930: // Query Input Value Occupancy
	IF (_bEnablePushButton) THEN
		fb301PushButton(	bInitialize := FALSE,
								bQueryInputValue := TRUE,
								bGetInputNotifications := FALSE,
								nShortAddress := nShortAddress,
								nInstanceNumber := 0);
		IF (NOT fb301PushButton.bReadingInputValue) THEN
			nPushBotton := fb301PushButton.nPushButtonEvent;
			nStep := 940;
			fb301PushButton(bInitialize := FALSE, bQueryInputValue := FALSE);
		END_IF
	ELSE
		nPushBotton := 1;
		nStep := 940;
	END_IF

940: // Query Input Value rotation direction
	IF (_bEnableRotation) THEN
		fb301Rotation(
			bInitialize:= FALSE, 
			nShortAddress:= nShortAddress, 
			nInstanceNumber:= 1, 
			bQueryInputValue:= TRUE, 
			bGetInputNotifications:= FALSE);	 
	
		IF (NOT fb301Rotation.bReadingInputValue) THEN
			nRotation := 4 ;//fb301Rotation.nPushButtonEvent; This are disabled, due to no data to query, before the device has being rotated
			nStep := 950;
			fb301Rotation(bQueryInputValue := FALSE);
		END_IF
	ELSE
		nRotation := 4;
		nStep := 950;
	END_IF

950: // Query Input actual position
	IF (_bEnablePosition) THEN
		fb302AbsoluteInputDevice(	bInitialize := FALSE,
							bQueryInputValue := TRUE,
							nShortAddress := nShortAddress,
							nInstanceNumber := 2,
							nResolution := 8);
		IF (NOT fb302AbsoluteInputDevice.bReadingInputValue) THEN
			nPosition := fb302AbsoluteInputDevice.nInputLevel;
			nStep := 0;
			fb302AbsoluteInputDevice(bInitialize := FALSE, bQueryInputValue := FALSE);
		END_IF
	ELSE
		nPosition := 0;
		nStep := 0;
	END_IF
{endregion}

ELSE
	nStep := 0;
END_CASE

THIS^.SetCommunication();
IF (THIS^.ParameterChanged()) THEN
	nErrorId := THIS^.CheckParameters();
	bError := (nErrorId > 0);
	IF (bError) THEN
		bParameterInvalid := TRUE;
		RETURN;
	ELSE
		bParameterInvalid := FALSE;
	END_IF
END_IF
IF (bParameterInvalid) THEN
	RETURN;
END_IF

{region 'Notifications'}
IF (NOT bInitializing) THEN
	rtrigReadingPushBotton(CLK := bQueryPushBotton);
	IF (rtrigReadingPushBotton.Q) THEN
		bReadingPushbotton:= TRUE;
	END_IF
	rtrigReadingRotation(CLK := bQueryRotation);
	IF (rtrigReadingRotation.Q) THEN
		bReadingRotation := TRUE;
	END_IF
	rtrigReadingPosition(CLK := bQueryPosition);
	IF (rtrigReadingPosition.Q) THEN
		bReadingPosition := TRUE;
	END_IF

	THIS^.SetCommunication();

	fb103ControlDevice(	bInitialize := FALSE,
						bGetPowerCycleNotifications := FALSE,
						nShortAddress := nShortAddress);
	rtrigError103Generic(CLK := fb103ControlDevice.bError);
	ftrigError103Generic(CLK := fb103ControlDevice.bError);
	IF (rtrigError103Generic.Q OR ftrigError103Generic.Q) THEN
		nErrorId := fb103ControlDevice.ipResultMessage.nEventId;
		bError := fb103ControlDevice.bError;
	END_IF

{region 'Pushbotton'}
	fb301PushButton(
		bInitialize:= FALSE, 
		nShortAddress:= nShortAddress, 
		nInstanceNumber:= 0, 
		bQueryInputValue:= bQueryPushBotton, 
		bGetInputNotifications:= TRUE);

	IF (bReadingPushbotton) THEN
		IF (NOT fb301PushButton.bReadingInputValue) THEN
			bReadingPushbotton := FALSE;
			IF (NOT fb301PushButton.bError) THEN
				nPushBotton := fb301PushButton.nPushButtonEvent;
			END_IF
		END_IF
	END_IF
	IF (NOT fb301PushButton.bError) THEN
		nPushBotton := fb301PushButton.nPushButtonEvent;
	END_IF
	rtrigError301PushButton(CLK := fb301PushButton.bError);
	ftrigError301PushButton(CLK := fb301PushButton.bError);
	IF (rtrigError301PushButton.Q OR ftrigError301PushButton.Q) THEN
		nErrorId := fb301PushButton.ipResultMessage.nEventId;
		bError := fb301PushButton.bError;
	END_IF
{endregion}

{region 'Rotation'}
	 
	fb301Rotation(
		bInitialize:= FALSE, 
		nShortAddress:= nShortAddress, 
		nInstanceNumber:= 1, 
		bQueryInputValue:= bQueryRotation, 
		bGetInputNotifications:= TRUE);	 		   
						 
	IF (bReadingRotation) THEN
		IF (NOT fb301Rotation.bReadingInputValue) THEN
			bReadingRotation := FALSE;
			IF (NOT fb301Rotation.bError) THEN
				nRotation := fb301Rotation.nPushButtonEvent;
			END_IF
		END_IF
	END_IF
	IF (NOT fb301Rotation.bError) THEN
		nRotation := fb301Rotation.nPushButtonEvent;
	END_IF
	rtrigError301Rotation(CLK := fb301Rotation.bError);
	ftrigError301Rotation(CLK := fb301Rotation.bError);
	IF (rtrigError301Rotation.Q OR ftrigError301Rotation.Q) THEN
		nErrorId := fb301Rotation.ipResultMessage.nEventId;
		bError := fb301Rotation.bError;
	END_IF
{endregion}

{region 'Position'}
	fb302AbsoluteInputDevice( bInitialize:= FALSE, 
						nShortAddress:= , 
						nInstanceNumber:= 2, 
						nResolution:= 8, 
						bQueryInputValue:= bQueryPosition, 
						bGetInputNotifications:= TRUE);

	IF (bReadingPosition) THEN
		IF (NOT fb302AbsoluteInputDevice.bReadingInputValue) THEN
			bReadingPosition := FALSE;
			IF (NOT fb302AbsoluteInputDevice.bError) THEN
				nPosition := fb302AbsoluteInputDevice.nInputLevel;
			END_IF
		END_IF
	END_IF
	IF (NOT fb302AbsoluteInputDevice.bError) THEN
		nPosition := fb302AbsoluteInputDevice.nInputLevel;
	END_IF
	rtrigError302AbsoluteInputDevice(CLK := fb302AbsoluteInputDevice.bError);
	ftrigError302AbsoluteInputDevice(CLK := fb302AbsoluteInputDevice.bError);
	IF (rtrigError302AbsoluteInputDevice.Q OR ftrigError302AbsoluteInputDevice.Q) THEN
		nErrorId := fb302AbsoluteInputDevice.ipResultMessage.nEventId;
		bError := fb302AbsoluteInputDevice.bError;
	END_IF
{endregion}
		  
END_IF
{endregion}

IF (bError) THEN
	nPushBotton := 1;
	nRotation := 4;
	nPosition := 0;
END_IF

IF nPushBotton.0 THEN
	bPressed := FALSE;
	bReleased:= TRUE;
END_IF
IF nPushBotton.1 THEN
	bPressed := TRUE;
	bReleased:= FALSE;
END_IF

IF nRotation.2 THEN
	bNeutral:= TRUE;
	bCCW := FALSE;
	bCW := FALSE;
ELSIF nRotation.0 THEN
	bNeutral:= FALSE;
	bCCW := FALSE;
	bCW := TRUE;
ELSIF nRotation.1 THEN
	bNeutral:= FALSE;
	bCCW := TRUE;
	bCW := FALSE;	
END_IF

stROTdata.bStopped:= bNeutral ;
stROTdata.bCW:= bCW ;
stROTdata.bCCW:= bCCW ;
stROTdata.bPressed:= bPressed ;
stROTdata.bReleased:= bReleased ;
stROTdata.nPos:= LWORD_TO_BYTE(nPosition) ;

// A TRUE at this input enables the instance for detecting movement. A FALSE at this input causes the sending of events from this instance to be disabled.
{attribute 'monitoring' := 'call'}
PROPERTY PUBLIC bEnablePosition : BOOL
GET
bEnablePosition := _bEnablePosition;
END_GET
SET
_bEnablePosition := bEnablePosition;
END_SET
END_PROPERTY

// Setting of the event priority (Low, MiddleLow, Middle, MiddleHigh).
{attribute 'monitoring' := 'call'}
PROPERTY PUBLIC eEventPriorityPosition : E_DALIEventPriority
GET
eEventPriorityPosition := _eEventPriorityPosition;
END_GET
SET
_eEventPriorityPosition := eEventPriorityPosition;
END_SET
END_PROPERTY

// Dead time (0...12750 ms) to ensure that not too many events are sent in succession. An event is only sent after expiry of the dead time timer. The dead time timer is restarted each time an event is sent.
{attribute 'monitoring' := 'call'}
PROPERTY PUBLIC nDeadtimerPosition : UINT
GET
nDeadtimerPosition := _nDeadtimeTimerPosition;
END_GET
SET
_nDeadtimeTimerPosition := nDeadtimerPosition;
END_SET
END_PROPERTY

// Time (0…255 s) after which the pending event of the measurement is repeated if no other event has occurred in the meantime.
{attribute 'monitoring' := 'call'}
PROPERTY PUBLIC nReportTimePosition : BYTE
GET
nReportTimePosition := _nReportTimerPosition;
END_GET
SET
_nReportTimerPosition := nReportTimePosition;
END_SET
END_PROPERTY

// A TRUE at this input enables the instance for measuring the brightness. A FALSE at this input causes the sending of events from this instance to be disabled.
{attribute 'monitoring' := 'call'}
PROPERTY PUBLIC bEnablePushButton : BOOL
GET
bEnablePushButton := _bEnablePushButton;
END_GET
SET
_bEnablePushButton := bEnablePushButton;
END_SET
END_PROPERTY

// Setting of the event priority (Low, MiddleLow, Middle, MiddleHigh).
{attribute 'monitoring' := 'call'}
PROPERTY PUBLIC eEventPriorityButton : E_DALIEventPriority
GET
eEventPriorityButton := _eEventPriorityPushButton;
END_GET
SET
_eEventPriorityPushButton := eEventPriorityButton;
END_SET
END_PROPERTY

// Deadtime (0...12750 ms), to ensure to send out an event until the deadtime timer has expired. The deadtime timer will be restarted every time an event is sent.
{attribute 'monitoring' := 'call'}
PROPERTY PUBLIC nDoubleTimerPushButton : UINT
GET
nDoubleTimerPushButton := _nDoubleTimerPushButton;
END_GET
SET
_nDoubleTimerPushButton := nDoubleTimerPushButton;
END_SET
END_PROPERTY

// Time (0...255 s) after which the pending event of the brightness sensor is repeated if no other event has occurred in the meantime.
{attribute 'monitoring' := 'call'}
PROPERTY PUBLIC nEventFilterPushButton : BYTE
GET
nEventFilterPushButton := _nEventFilterPushButton;
END_GET
SET
_nEventFilterPushButton := nEventFilterPushButton;
END_SET
END_PROPERTY

// Value (0...25 %) for calculating a hysteresis value in order to prevent frequent and disturbing changes when measuring the brightness.
{attribute 'monitoring' := 'call'}
PROPERTY PUBLIC nRepeatTimerPushButton : uint
GET
nRepeatTimerPushButton := _nRepeatTimerPushButton;
END_GET
SET
_nRepeatTimerPushButton := nRepeatTimerPushButton;
END_SET
END_PROPERTY

// As the percentage hysteresis can also lead to large fluctuations at low brightness, a minimum hysteresis (0...255) can be specified with this variable.
{attribute 'monitoring' := 'call'}
PROPERTY PUBLIC nShortTimerPushButton : UINT
GET
nShortTimerPushButton := _nShortTimerPushButton;
END_GET
SET
_nShortTimerPushButton := nShortTimerPushButton;
END_SET
END_PROPERTY

// Time (0...255 s) after which the pending event of the brightness sensor is repeated if no other event has occurred in the meantime.
{attribute 'monitoring' := 'call'}
PROPERTY PUBLIC nStuckTimerPushButton : BYTE
GET
nStuckTimerPushButton := _nStuckTimerPushButton;
END_GET
SET
_nStuckTimerPushButton := nStuckTimerPushButton;
END_SET
END_PROPERTY

// A TRUE at this input enables the instance for detecting movement. A FALSE at this input causes the sending of events from this instance to be disabled.
{attribute 'monitoring' := 'call'}
PROPERTY PUBLIC bEnableRotation : BOOL
GET
bEnableRotation := _bEnableRotation;
END_GET
SET
_bEnableRotation := bEnableRotation;
END_SET
END_PROPERTY

// Setting of the event priority (Low, MiddleLow, Middle, MiddleHigh).
{attribute 'monitoring' := 'call'}
PROPERTY PUBLIC eEventPriorityRotation : E_DALIEventPriority
GET
eEventPriorityRotation := _eEventPriorityRotation;
END_GET
SET
_eEventPriorityRotation := eEventPriorityRotation;
END_SET
END_PROPERTY

// Setting of the event filter.
{attribute 'monitoring' := 'call'}
PROPERTY PUBLIC nEventFilterRotation : byte
GET
nEventFilterRotation := _nEventFilterRotation;
END_GET
SET
_nEventFilterRotation:= nEventFilterRotation;
END_SET
END_PROPERTY

// Checks whether all parameters are valid.
// Return codes:
//   0: no error.
//	 1..999: error codes of the library
//   1000... : custom error codes
METHOD PRIVATE CheckParameters : UDINT
CheckParameters := 0;
IF (_ipDALICommunication = 0) THEN
	CheckParameters := TC_EVENTS.TcDALIEventClass.TheInterfaceToTheCommunicationBufferIsNotInitialized.nEventId;
ELSIF (nShortAddress > 63) THEN
	CheckParameters := TC_EVENTS.TcDALIEventClass.ParameterShortAddressLiesOutsideOfTheValidRange2.nEventId;
{region 'Botton'}
ELSIF (_nDoubleTimerPushButton > 2000) THEN
	CheckParameters := TC_EVENTS.TcDALIEventClass.ParameterDoubleTimerPart301LiesOutsideOfTheValidRange.nEventId;
ELSIF ((_nRepeatTimerPushButton < 100) OR (_nRepeatTimerPushButton > 2000)) THEN
	CheckParameters := TC_EVENTS.TcDALIEventClass.ParameterRepeatTimerLiesOutsideOfTheValidRange.nEventId;
ELSIF (nShortTimerPushButton > 5100) THEN
	CheckParameters := TC_EVENTS.TcDALIEventClass.ParameterShortTimerPart301LiesOutsideOfTheValidRange.nEventId;
ELSIF ((_nStuckTimerPushButton < 5) OR (_nStuckTimerPushButton > 255)) THEN
	CheckParameters := TC_EVENTS.TcDALIEventClass.ParameterStuckTimerPart301LiesOutsideOfTheValidRange.nEventId;
ELSIF ((_eEventPriorityPushButton <> E_DALIEventPriority.Low) AND (_eEventPriorityPushButton <> E_DALIEventPriority.MiddleLow) AND
       (_eEventPriorityPushButton <> E_DALIEventPriority.Middle) AND (_eEventPriorityPushButton <> E_DALIEventPriority.MiddleHigh)) THEN
	CheckParameters := TC_EVENTS.TcDALIEventClass.ParameterEventPriorityDeviceLiesOutsideOfTheValidRange.nEventId;
{endregion}
{region 'Rotation'}
ELSIF ((_eEventPriorityRotation <> E_DALIEventPriority.Low) AND (_eEventPriorityRotation <> E_DALIEventPriority.MiddleLow) AND
       (_eEventPriorityRotation <> E_DALIEventPriority.Middle) AND (_eEventPriorityRotation <> E_DALIEventPriority.MiddleHigh)) THEN
	CheckParameters := TC_EVENTS.TcDALIEventClass.ParameterEventPriorityDeviceLiesOutsideOfTheValidRange.nEventId;
{endregion}
{region 'Position'}
ELSIF (_nDeadtimeTimerPosition > 12750) THEN
	CheckParameters := TC_EVENTS.TcDALIEventClass.ParameterDeadtimeTimerPart302LiesOutsideOfTheValidRange.nEventId;
ELSIF ((_eEventPriorityPosition <> E_DALIEventPriority.Low) AND (_eEventPriorityPosition <> E_DALIEventPriority.MiddleLow) AND
       (_eEventPriorityPosition <> E_DALIEventPriority.Middle) AND (_eEventPriorityPosition <> E_DALIEventPriority.MiddleHigh)) THEN
	CheckParameters := TC_EVENTS.TcDALIEventClass.ParameterEventPriorityDeviceLiesOutsideOfTheValidRange.nEventId;
{endregion}
//ELSIF (check your parameter) THEN
//	CheckParameters := 1000;
//ELSIF (check another parameter) THEN
//	CheckParameters := 1001;
END_IF
END_METHOD

METHOD FB_init : BOOL
VAR_INPUT
	bInitRetains			:	BOOL; // if TRUE, the retain variables are initialized (warm start / cold start)
	bInCopyCode				:	BOOL;  // if TRUE, the instance afterwards gets moved into the copy code (online change)
	ipDALICommunication 	:	I_DALICommunication;
END_VAR
_ipDALICommunication := ipDALICommunication;
END_METHOD

// Property to set the referenz to the communication function block.
{attribute 'monitoring' := 'call'}
PROPERTY PUBLIC ipDALICommunication : I_DALICommunication
GET
ipDALICommunication := _ipDALICommunication;
END_GET
SET
_ipDALICommunication := ipDALICommunication;
END_SET
END_PROPERTY

// Return codes:
//   FALSE: no change
//   TRUE: parameter are changed
{attribute 'hide'}
METHOD PRIVATE ParameterChanged : BOOL
VAR_INPUT
END_VAR
IF (nShortAddress <> nShortAddressCheck) THEN
	ParameterChanged := TRUE;
	nShortAddressCheck := nShortAddress;
ELSE
	ParameterChanged := FALSE;
END_IF
END_METHOD

// Apply the preset value of IpDALICommunication if available.
METHOD PRIVATE SetCommunication : BOOL
VAR_INPUT
END_VAR
fb103ControlDevice.ipDALICommunication := THIS^.ipDALICommunication;
fb301PushButton.ipDALICommunication := THIS^.ipDALICommunication;
fb301Rotation.ipDALICommunication := THIS^.ipDALICommunication;
fb302AbsoluteInputDevice.ipDALICommunication := THIS^.ipDALICommunication;
fbSavePersistentVariables.ipDALICommunication := THIS^.ipDALICommunication;
fbStartQuiescentMode.ipDALICommunication := THIS^.ipDALICommunication;
fbStopQuiescentMode.ipDALICommunication := THIS^.ipDALICommunication;
END_METHOD

END_FUNCTION_BLOCK

// POUs/DALI/DALI_Devices/Lunatone/FB_DALI_LunatoneMC
FUNCTION_BLOCK FB_DALI_LunatoneMC
VAR_INPUT
	byShrtAdr				: BYTE;
	bInitialize				: BOOL := TRUE;
	ipCommunication			: I_DALICommunication;
	DALI_LINE_NUM			: INT := 1;	
	stLunatoneMCSetup		: ST_LunatoneMCSetup;		
END_VAR
VAR_OUTPUT
	arrButtons				: ARRAY [1..4] OF ST_DALIButton;
END_VAR
		
VAR
	fbButtons 				: FB_DALI_Lunatone_MC(0) ;

	arrQueryInput 			: ARRAY [1..4] OF BOOL;
	arrReadingInput 		: ARRAY [1..4] OF BOOL;
	arrPushButtonEvent 		: ARRAY [1..4] OF WORD; (* Bit 0 - Push button released.
									 Bit 1 - Push button pressed..
									 Bit 2 - Short keystroke.
									 Bit 3 - Double keystroke.
									 Bit 4 - Start long keystroke.
									 Bit 5 - Repeat long keystroke.
									 Bit 6 - Stop long keystroke.
									 Bit 7 - Push button free again; was previously blocked.
									 Bit 8 - Push button blocked. *)

	fbDelaySetupDALIDevice	: TON;
	tDelayTime				: TIME;
	bInitSensor				: BOOL;
	fbInitDone				: F_TRIG;
	bInitDone				: BOOL;
	bInitErr				: BOOL;
	bInitializing			: BOOL;
	bInitTimeOut			: BOOL;
	fbInitTimeOut			: TON;
END_VAR

fbButtons.ipDALICommunication:= ipCommunication ;

	fbButtons.bEnablePushButton1:= stLunatoneMCSetup.arrEnablePushButton[1];
	fbButtons.bEnablePushButton2:= stLunatoneMCSetup.arrEnablePushButton[2];
	fbButtons.bEnablePushButton3:= stLunatoneMCSetup.arrEnablePushButton[3];
	fbButtons.bEnablePushButton4:= stLunatoneMCSetup.arrEnablePushButton[4];
	
	fbButtons.eEventPriorityPushButton1:= stLunatoneMCSetup.arrEventPriorityPushButton[1];
	fbButtons.eEventPriorityPushButton2:= stLunatoneMCSetup.arrEventPriorityPushButton[2];
	fbButtons.eEventPriorityPushButton3:= stLunatoneMCSetup.arrEventPriorityPushButton[3];
	fbButtons.eEventPriorityPushButton4:= stLunatoneMCSetup.arrEventPriorityPushButton[4];

	fbButtons.nDoubleTimerPushButton1 := stLunatoneMCSetup.nDoubleTimerPushButton;
	fbButtons.nDoubleTimerPushButton2:= stLunatoneMCSetup.nDoubleTimerPushButton;
	fbButtons.nDoubleTimerPushButton3:= stLunatoneMCSetup.nDoubleTimerPushButton;
	fbButtons.nDoubleTimerPushButton4:= stLunatoneMCSetup.nDoubleTimerPushButton;
	
	fbButtons.nEventFilterPushButton1 :=stLunatoneMCSetup.nEventFilterPushButton[1] ;
	fbButtons.nEventFilterPushButton2 :=stLunatoneMCSetup.nEventFilterPushButton[2] ;
	fbButtons.nEventFilterPushButton3 :=stLunatoneMCSetup.nEventFilterPushButton[3] ;
	fbButtons.nEventFilterPushButton4 :=stLunatoneMCSetup.nEventFilterPushButton[4] ;
	
	fbButtons.nRepeatTimerPushButton1 := stLunatoneMCSetup.nRepeatTimerPushButton;
	fbButtons.nRepeatTimerPushButton2 := stLunatoneMCSetup.nRepeatTimerPushButton;
	fbButtons.nRepeatTimerPushButton3 := stLunatoneMCSetup.nRepeatTimerPushButton;
	fbButtons.nRepeatTimerPushButton4 := stLunatoneMCSetup.nRepeatTimerPushButton;
	
	fbButtons.nShortTimerPushButton1 := stLunatoneMCSetup.nShortTimerPushButton ;
	fbButtons.nShortTimerPushButton2 := stLunatoneMCSetup.nShortTimerPushButton ;
	fbButtons.nShortTimerPushButton3 := stLunatoneMCSetup.nShortTimerPushButton ;
	fbButtons.nShortTimerPushButton4 := stLunatoneMCSetup.nShortTimerPushButton ;
	
	fbButtons.nStuckTimerPushButton1 := stLunatoneMCSetup.nStuckTimerPushButton ;
	fbButtons.nStuckTimerPushButton2 := stLunatoneMCSetup.nStuckTimerPushButton ;
	fbButtons.nStuckTimerPushButton3 := stLunatoneMCSetup.nStuckTimerPushButton ;
	fbButtons.nStuckTimerPushButton4 := stLunatoneMCSetup.nStuckTimerPushButton ;

//Calculate delay time for init sensor
tDelayTime := INT_TO_TIME((BYTE_TO_INT(byShrtAdr) * 400));	
fbDelaySetupDALIDevice(IN:= bInitialize , PT:=tDelayTime , Q=> , ET=> );	
	
IF fbDelaySetupDALIDevice.q AND NOT GVL_DALI.arrbBlockDTR[DALI_LINE_NUM] AND NOT (bInitDone OR bInitErr) THEN
	bInitDone := FALSE;
	bInitErr := FALSE;
	bInitSensor:= TRUE;
	GVL_DALI.arrbBlockDTR[DALI_LINE_NUM]:= TRUE;
END_IF

fbButtons(
	bError=> , 
	ipResultMessage=> , 
	bInitialize:= bInitSensor , 
	nShortAddress:= byShrtAdr, 
	nOptions:= , 
	bQueryInputValue1:= arrQueryInput[1], 
	bQueryInputValue2:= arrQueryInput[2], 
	bQueryInputValue3:= arrQueryInput[3], 
	bQueryInputValue4:= arrQueryInput[4], 
	bInitializing=> bInitializing, 
	bReadingInputValue1=> arrReadingInput[1] , 
	bReadingInputValue2=> arrReadingInput[2] , 
	bReadingInputValue3=> arrReadingInput[3] , 
	bReadingInputValue4=> arrReadingInput[4] , 
	nPushButton1Event=> arrPushButtonEvent[1], 
	nPushButton2Event=> arrPushButtonEvent[2], 
	nPushButton3Event=> arrPushButtonEvent[3], 
	nPushButton4Event=> arrPushButtonEvent[4]
);	
fbInitDone(CLK:=bInitSensor AND bInitializing );	
	IF fbInitDone.Q THEN
		IF NOT bInitTimeOut THEN
			bInitDone := TRUE;
			bInitErr := FALSE;
			GVL_DALI.arrbBlockDTR[DALI_LINE_NUM]:= FALSE;
		ELSE
			bInitErr := TRUE;
			GVL_DALI.arrbBlockDTR[DALI_LINE_NUM]:= FALSE;
		END_IF
	END_IF

fbInitTimeOut(IN:=bInitializing, PT:= T#15S); 

IF fbInitTimeOut.Q THEN
	bInitErr := TRUE;
	GVL_DALI.arrbBlockDTR[DALI_LINE_NUM]:= FALSE;
END_IF


IF NOT bInitialize THEN
		fbInitTimeOut(IN:= FALSE);
		bInitSensor:= FALSE;
		bInitDone := FALSE;
		bInitErr := FALSE;
END_IF	
	A_Sort_Event_Button1();
	A_Sort_Event_Button2();
	A_Sort_Event_Button3();
	A_Sort_Event_Button4();

ACTION A_Sort_Event_Button1:
IF arrPushButtonEvent[1].1 THEN
	arrButtons[1].bPressed:= TRUE;
	arrButtons[1].bReleased:= FALSE;
END_IF

IF arrPushButtonEvent[1].0 THEN
	arrButtons[1].bPressed:= FALSE;
	arrButtons[1].bReleased:= TRUE;
END_IF

IF arrPushButtonEvent[1].2 THEN
	arrButtons[1].bShortPress:= TRUE;
END_IF

IF arrPushButtonEvent[1].3 THEN
	arrButtons[1].bDoublePress:= TRUE;
END_IF

IF arrPushButtonEvent[1].4 THEN
	arrButtons[1].bLongPressStop:= FALSE;
	arrButtons[1].bLongPressStart:= TRUE;
	arrButtons[1].bLongPressRepeat:= FALSE;	
END_IF

arrButtons[1].bLongPressRepeat:= arrPushButtonEvent[1].5 ;

IF arrPushButtonEvent[1].6 THEN
	arrButtons[1].bLongPressStop:= TRUE;
	arrButtons[1].bLongPressStart:= FALSE;
	arrButtons[1].bLongPressRepeat:= FALSE;	
END_IF

IF arrPushButtonEvent[1].7 THEN
	arrButtons[1].bPressed:= FALSE;
	arrButtons[1].bReleased:= FALSE;
	arrButtons[1].bShortPress:= FALSE;
	arrButtons[1].bDoublePress:= FALSE;	
	arrButtons[1].bLongPressStart:= FALSE;
	arrButtons[1].bLongPressRepeat:= FALSE;	
	arrButtons[1].bLongPressStop:= FALSE;	
	arrButtons[1].bButtonFree := TRUE;
END_IF
END_ACTION

ACTION A_Sort_Event_Button2:

IF arrPushButtonEvent[2].1 THEN
	arrButtons[2].bPressed:= TRUE;
	arrButtons[2].bReleased:= FALSE;
END_IF

IF arrPushButtonEvent[2].0 THEN
	arrButtons[2].bPressed:= FALSE;
	arrButtons[2].bReleased:= TRUE;
END_IF

IF arrPushButtonEvent[2].2 THEN
	arrButtons[2].bShortPress:= TRUE;
END_IF

IF arrPushButtonEvent[2].3 THEN
	arrButtons[2].bDoublePress:= TRUE;
END_IF

IF arrPushButtonEvent[2].4 THEN
	arrButtons[2].bLongPressStop:= FALSE;
	arrButtons[2].bLongPressStart:= TRUE;
	arrButtons[2].bLongPressRepeat:= FALSE;	
END_IF

arrButtons[2].bLongPressRepeat:= arrPushButtonEvent[2].5 ;

IF arrPushButtonEvent[2].6 THEN
	arrButtons[2].bLongPressStop:= TRUE;
	arrButtons[2].bLongPressStart:= FALSE;
	arrButtons[2].bLongPressRepeat:= FALSE;	
END_IF

IF arrPushButtonEvent[2].7 THEN
	arrButtons[2].bPressed:= FALSE;
	arrButtons[2].bReleased:= FALSE;
	arrButtons[2].bShortPress:= FALSE;
	arrButtons[2].bDoublePress:= FALSE;	
	arrButtons[2].bLongPressStart:= FALSE;
	arrButtons[2].bLongPressRepeat:= FALSE;	
	arrButtons[2].bLongPressStop:= FALSE;	
	arrButtons[2].bButtonFree := TRUE;
END_IF
END_ACTION

ACTION A_Sort_Event_Button3:

IF arrPushButtonEvent[3].1 THEN
	arrButtons[3].bPressed:= TRUE;
	arrButtons[3].bReleased:= FALSE;
END_IF

IF arrPushButtonEvent[3].0 THEN
	arrButtons[3].bPressed:= FALSE;
	arrButtons[3].bReleased:= TRUE;
END_IF

IF arrPushButtonEvent[3].2 THEN
	arrButtons[3].bShortPress:= TRUE;
END_IF

IF arrPushButtonEvent[3].3 THEN
	arrButtons[3].bDoublePress:= TRUE;
END_IF

IF arrPushButtonEvent[3].4 THEN
	arrButtons[3].bLongPressStop:= FALSE;
	arrButtons[3].bLongPressStart:= TRUE;
	arrButtons[3].bLongPressRepeat:= FALSE;	
END_IF

arrButtons[3].bLongPressRepeat:= arrPushButtonEvent[3].5 ;

IF arrPushButtonEvent[3].6 THEN
	arrButtons[3].bLongPressStop:= TRUE;
	arrButtons[3].bLongPressStart:= FALSE;
	arrButtons[3].bLongPressRepeat:= FALSE;	
END_IF

IF arrPushButtonEvent[3].7 THEN
	arrButtons[3].bPressed:= FALSE;
	arrButtons[3].bReleased:= FALSE;
	arrButtons[3].bShortPress:= FALSE;
	arrButtons[3].bDoublePress:= FALSE;	
	arrButtons[3].bLongPressStart:= FALSE;
	arrButtons[3].bLongPressRepeat:= FALSE;	
	arrButtons[3].bLongPressStop:= FALSE;	
	arrButtons[3].bButtonFree := TRUE;
END_IF
END_ACTION

ACTION A_Sort_Event_Button4:

IF arrPushButtonEvent[4].1 THEN
	arrButtons[4].bPressed:= TRUE;
	arrButtons[4].bReleased:= FALSE;
END_IF

IF arrPushButtonEvent[4].0 THEN
	arrButtons[4].bPressed:= FALSE;
	arrButtons[4].bReleased:= TRUE;
END_IF

IF arrPushButtonEvent[4].2 THEN
	arrButtons[4].bShortPress:= TRUE;
END_IF

IF arrPushButtonEvent[4].3 THEN
	arrButtons[4].bDoublePress:= TRUE;
END_IF

IF arrPushButtonEvent[4].4 THEN
	arrButtons[4].bLongPressStop:= FALSE;
	arrButtons[4].bLongPressStart:= TRUE;
	arrButtons[4].bLongPressRepeat:= FALSE;	
END_IF

arrButtons[4].bLongPressRepeat:= arrPushButtonEvent[4].5 ;

IF arrPushButtonEvent[4].6 THEN
	arrButtons[4].bLongPressStop:= TRUE;
	arrButtons[4].bLongPressStart:= FALSE;
	arrButtons[4].bLongPressRepeat:= FALSE;	
END_IF

IF arrPushButtonEvent[4].7 THEN
	arrButtons[4].bPressed:= FALSE;
	arrButtons[4].bReleased:= FALSE;
	arrButtons[4].bShortPress:= FALSE;
	arrButtons[4].bDoublePress:= FALSE;	
	arrButtons[4].bLongPressStart:= FALSE;
	arrButtons[4].bLongPressRepeat:= FALSE;	
	arrButtons[4].bLongPressStop:= FALSE;	
	arrButtons[4].bButtonFree := TRUE;
END_IF
END_ACTION

END_FUNCTION_BLOCK

// POUs/DALI/DALI_Devices/NIKO/FB_NIKO_P46xx_10Pcs
FUNCTION_BLOCK FB_NIKO_P46xx_10Pcs
VAR_INPUT
	arrShrtAdr					: ARRAY [1..10] OF BYTE;
	bInitialize					: BOOL := TRUE;
	ipCommunication				: I_DALICommunication;
	DALI_LINE_NUM				: INT := 1;	
END_VAR
VAR_OUTPUT
	arrInitErr: ARRAY [1.. nNumberOfSensors] OF BOOL;
	arrInitDone: ARRAY [1.. nNumberOfSensors] OF BOOL;
END_VAR
VAR
	arrNiko_P46xx				: ARRAY [1.. nNumberOfSensors] OF FB_DALI_Niko_P46LR(0);
	
	arrDelaySetupDALIDevice		: ARRAY [1.. nNumberOfSensors] Of TON;
	arrtDelayTime				: ARRAY [1.. nNumberOfSensors] OF TIME;
	arrInitSensor				: ARRAY [1.. nNumberOfSensors] OF BOOL;
	arrInitDone_FTrig			: ARRAY [1.. nNumberOfSensors] OF F_TRIG;
	arrInitializing				: ARRAY [1.. nNumberOfSensors] OF BOOL;
	bQueryBrightness 			: BOOL;
	bQueryOccupancy				: BOOL;
	eEventPriorityOccupancy		: E_DALIEventPriority := E_DALIEVENTPRIORITY.Middle;
	nHoldTimerOccupancy			: WORD := 5; // Value in s. 	
	nReportTimerOccupancy		: BYTE := 120; // Value in s, Preset manufacturer value
	nDeadtimeTimerOccupancy		: WORD := 100; // Value in ms, Predefined Value of DALI Standard
	bCancelHoldTimerOccupancy	: BOOL;
	nSensitivityOccupancy		: BYTE:= 3; //setting Sensivity (0..4) 0 (Off), 1 (Min), 2(Low), 3(High) and 4 (Max)

	bEnableLuxEvent				: BOOL;
	eEventPriorityBrightness	: E_DALIEventPriority := E_DALIEVENTPRIORITY.Middle;
	nDeadtimeTimerBrightness	: WORD := 1500; // Value in ms, Predefined Value of DALI Standard
	nHysteresisBrightness		: BYTE := 2; // Value in %
	nHysteresisMinBrightness	: BYTE := 10; // Absolute Value, depending on the manufacturer specific resolution
	nReportTimerBrightness		: BYTE := 120; // Value in s, Preset manufacturer value

	bAutoRead					: BOOL;
	fbAutoRequestBrightness_TON	: TOF;
	bInitTimeOut				: BOOL;
	fbInitTimeOut				: ARRAY [1.. nNumberOfSensors] OF TON;
	nIdxScan					: BYTE;
	nPirIdxOn					: BYTE;
	nBrightnessIdx				: BYTE;
	fBrightness_1				: REAL;
	fBrightness_2				: REAL;
	fBrightness_3				: REAL;
	fBrightness_4				: REAL;
	fBrightness_5				: REAL;
	fBrightness_6				: REAL;
	fBrightness_7				: REAL;
	fBrightness_8				: REAL;
	fBrightness_9				: REAL;
	fBrightness_10				: REAL;
	bInitDone					: BOOL;
	bInitScalesDone				: BOOL;
	
	nCheckIdx: INT;
END_VAR
VAR_IN_OUT
	stSensorSetup 				: ST_DALI_NIKOP46SetupData ;	
	stPirSensorData				: ST_DALI_Sensor;
	arrSensorScales				: ARRAY [1.. 10] OF ST_DALI_SensorScaleMode;
END_VAR

VAR CONSTANT
	nNumberOfSensors: BYTE := 10;
END_VAR


arrNiko_P46xx[1].ipDALICommunication := ipCommunication;
arrNiko_P46xx[2].ipDALICommunication := ipCommunication;
arrNiko_P46xx[3].ipDALICommunication := ipCommunication;
arrNiko_P46xx[4].ipDALICommunication := ipCommunication;
arrNiko_P46xx[5].ipDALICommunication := ipCommunication;
arrNiko_P46xx[6].ipDALICommunication := ipCommunication;
arrNiko_P46xx[7].ipDALICommunication := ipCommunication;
arrNiko_P46xx[8].ipDALICommunication := ipCommunication;
arrNiko_P46xx[9].ipDALICommunication := ipCommunication;
arrNiko_P46xx[10].ipDALICommunication := ipCommunication;

IF NOT bInitScalesDone THEN
	FOR nCheckIdx:= 1 TO 10 DO
		IF arrSensorScales[nCheckIdx].fMeassureMaxSensor = 0 THEN
			arrSensorScales[nCheckIdx].fMeassureMaxSensor := 1;
		END_IF
		IF arrSensorScales[nCheckIdx].fReadMaxSensor = 0 THEN
			arrSensorScales[nCheckIdx].fReadMaxSensor := 1;
		END_IF
	END_FOR
	bInitScalesDone := TRUE;
END_IF

IF ipCommunication <> 0 THEN
	A_NIKO_P46xx();
END_IF

ACTION A_NIKO_P46xx:


FOR nIdxScan := 1 TO nNumberOfSensors DO
	//Setup parameters
		//Setup Motion part of sensor (Instance 0)
		arrNiko_P46xx[nIdxScan].eEventPriorityOccupancy:= stSensorSetup.eEventPriorityOccupancy;
		arrNiko_P46xx[nIdxScan].nHoldTimerOccupancy := stSensorSetup.nHoldTimerOccupancy ;
		arrNiko_P46xx[nIdxScan].nReportTimerOccupancy := stSensorSetup.nReportTimerOccupancy;
		arrNiko_P46xx[nIdxScan].nDeadtimeTimerOccupancy:= stSensorSetup.nDeadtimeTimerOccupancy;
		arrNiko_P46xx[nIdxScan].nSensitivityOccupancyA:= stSensorSetup.nSensitivityPIRSegmentA;
		arrNiko_P46xx[nIdxScan].nSensitivityOccupancyB:= stSensorSetup.nSensitivityPIRSegmentB;
		arrNiko_P46xx[nIdxScan].nSensitivityOccupancyC:= stSensorSetup.nSensitivityPIRSegmentC;
	
		//Setup Brightness part of sensor (Instance 1)
		arrNiko_P46xx[nIdxScan].bEnableBrightness := stSensorSetup.bEnableInstanceBrightness;
		arrNiko_P46xx[nIdxScan].eEventPriorityBrightness:= stSensorSetup.eEventPriorityBrightness;
		arrNiko_P46xx[nIdxScan].nDeadtimeTimerBrightness:= stSensorSetup.nDeadtimeTimerBrightness;
		arrNiko_P46xx[nIdxScan].nHysteresisBrightness:= stSensorSetup.nHysteresisBrightness;
		arrNiko_P46xx[nIdxScan].nHysteresisMinBrightness:= stSensorSetup.nHysteresisMinBrightness;
		arrNiko_P46xx[nIdxScan].nReportTimerBrightness:= stSensorSetup.nReportTimerBrightness;
		
	//Calculate delay time for init sensor
	arrtDelayTime[nIdxScan] := INT_TO_TIME((BYTE_TO_INT(arrShrtAdr[nIdxScan]) * 400));	
	arrDelaySetupDALIDevice[nIdxScan](IN:= bInitialize , PT:=arrtDelayTime[nIdxScan] , Q=> , ET=> );	
		
	IF arrDelaySetupDALIDevice[nIdxScan].q AND NOT GVL_DALI.arrbBlockDTR[DALI_LINE_NUM] AND NOT (arrInitDone[nIdxScan] OR arrInitErr[nIdxScan]) THEN
		arrInitSensor[nIdxScan]:= TRUE;
		GVL_DALI.arrbBlockDTR[DALI_LINE_NUM]:= TRUE;
	END_IF
	
	bQueryBrightness:= stPirSensorData.bQueryBrightness OR NOT bAutoRead;
	
	fbAutoRequestBrightness_TON(IN:= NOT fbAutoRequestBrightness_TON.Q  AND NOT stPirSensorData.bQueryBrightness , PT:= (arrtDelayTime[nIdxScan] + T#12M) , Q=>bAutoRead , ET=> );
	
	bQueryOccupancy:= NOT bAutoRead OR stPirSensorData.bQueryBrightness;
	
	arrNiko_P46xx[nIdxScan](
		bError=> , 
		ipResultMessage=> , 
		bInitialize:=  arrInitSensor[nIdxScan], 
		nShortAddress:= arrShrtAdr[nIdxScan], 
		nOptions:= , 
		bQueryOccupancy:= bQueryOccupancy, 
		bQueryBrightness:= bQueryBrightness, 
		bCancelHoldTimerOccupancy:= bCancelHoldTimerOccupancy, 
		bInitializing=> arrInitializing[nIdxScan] , 
		bReadingOccupancy=> , 
		bReadingBrightness=> , 
		bOccupied=> , 
		nBrightnessLevel=> );
	
	IF arrNiko_P46xx[nIdxScan].bError THEN
		GVL_DALI_LatestError.arrLineShrtAddr[DALI_LINE_NUM] :=arrShrtAdr[nIdxScan];
	END_IF
	
	arrInitDone_FTrig[nIdxScan](CLK:=arrInitializing[nIdxScan] );	
		IF arrInitDone_FTrig[nIdxScan].Q THEN
			IF NOT bInitTimeOut THEN
				arrInitDone[nIdxScan] := TRUE;
				GVL_DALI.arrbBlockDTR[DALI_LINE_NUM]:= FALSE;
			ELSE
				arrInitErr[nIdxScan] := TRUE;
				GVL_DALI.arrbBlockDTR[DALI_LINE_NUM]:= FALSE;
			END_IF
		END_IF
		
	fbInitTimeOut[nIdxScan](IN:=arrInitSensor[nIdxScan] AND NOT arrInitDone[nIdxScan], PT:= T#10S); 
	
	IF fbInitTimeOut[nIdxScan].Q THEN
		arrInitErr[nIdxScan] := TRUE;
		GVL_DALI.arrbBlockDTR[DALI_LINE_NUM]:= FALSE;
	END_IF
END_FOR

stPirSensorData.bPrc:= FALSE;
FOR nPirIdxOn:= 1 TO nNumberOfSensors DO
	IF arrNiko_P46xx[nPirIdxOn].bOccupied THEN
		stPirSensorData.bPrc:= TRUE;
		EXIT;
	END_IF
END_FOR

stPirSensorData.bBrightnessRead:=	arrNiko_P46xx[1].bReadingBrightness OR arrNiko_P46xx[2].bReadingBrightness OR arrNiko_P46xx[3].bReadingBrightness OR arrNiko_P46xx[4].bReadingBrightness OR arrNiko_P46xx[5].bReadingBrightness OR
														arrNiko_P46xx[6].bReadingBrightness OR arrNiko_P46xx[7].bReadingBrightness OR arrNiko_P46xx[8].bReadingBrightness OR arrNiko_P46xx[9].bReadingBrightness OR arrNiko_P46xx[10].bReadingBrightness;

fBrightness_1:= F_fScale(0, arrSensorScales[1].fReadMaxSensor, 0, arrSensorScales[1].fMeassureMaxSensor, 0, arrNiko_P46xx[1].nBrightnessLevel);
fBrightness_2:= F_fScale(0, arrSensorScales[2].fReadMaxSensor, 0, arrSensorScales[2].fMeassureMaxSensor, 0, arrNiko_P46xx[2].nBrightnessLevel);
fBrightness_3:= F_fScale(0, arrSensorScales[3].fReadMaxSensor, 0, arrSensorScales[3].fMeassureMaxSensor, 0, arrNiko_P46xx[3].nBrightnessLevel);
fBrightness_4:= F_fScale(0, arrSensorScales[4].fReadMaxSensor, 0, arrSensorScales[4].fMeassureMaxSensor, 0, arrNiko_P46xx[4].nBrightnessLevel);
fBrightness_5:= F_fScale(0, arrSensorScales[5].fReadMaxSensor, 0, arrSensorScales[5].fMeassureMaxSensor, 0, arrNiko_P46xx[5].nBrightnessLevel);
fBrightness_6:= F_fScale(0, arrSensorScales[6].fReadMaxSensor, 0, arrSensorScales[6].fMeassureMaxSensor, 0, arrNiko_P46xx[6].nBrightnessLevel);
fBrightness_7:= F_fScale(0, arrSensorScales[7].fReadMaxSensor, 0, arrSensorScales[7].fMeassureMaxSensor, 0, arrNiko_P46xx[7].nBrightnessLevel);
fBrightness_8:= F_fScale(0, arrSensorScales[8].fReadMaxSensor, 0, arrSensorScales[8].fMeassureMaxSensor, 0, arrNiko_P46xx[8].nBrightnessLevel);
fBrightness_9:= F_fScale(0, arrSensorScales[9].fReadMaxSensor, 0, arrSensorScales[9].fMeassureMaxSensor, 0, arrNiko_P46xx[9].nBrightnessLevel);
fBrightness_10:= F_fScale(0, arrSensorScales[10].fReadMaxSensor, 0, arrSensorScales[10].fMeassureMaxSensor, 0, arrNiko_P46xx[10].nBrightnessLevel);

IF fBrightness_1 <> 0 THEN
	stPirSensorData.fBrightness:= fBrightness_1;
END_IF
IF fBrightness_2 <> 0 THEN
	stPirSensorData.fBrightness:= MIN(fBrightness_2, stPirSensorData.fBrightness);
END_IF
IF fBrightness_3 <> 0 THEN
	stPirSensorData.fBrightness:=  MIN(fBrightness_3, stPirSensorData.fBrightness);
END_IF
IF fBrightness_4 <> 0 THEN
	stPirSensorData.fBrightness:=  MIN(fBrightness_4, stPirSensorData.fBrightness);
END_IF
IF fBrightness_5 <> 0 THEN
	stPirSensorData.fBrightness:=  MIN(fBrightness_5, stPirSensorData.fBrightness);
END_IF
IF fBrightness_6 <> 0 THEN
	stPirSensorData.fBrightness:= MIN(fBrightness_6, stPirSensorData.fBrightness);
END_IF
IF fBrightness_7 <> 0 THEN
	stPirSensorData.fBrightness:=  MIN(fBrightness_7, stPirSensorData.fBrightness);
END_IF
IF fBrightness_8 <> 0 THEN
	stPirSensorData.fBrightness:=  MIN(fBrightness_8, stPirSensorData.fBrightness);
END_IF
IF fBrightness_9 <> 0 THEN
	stPirSensorData.fBrightness:=  MIN(fBrightness_9, stPirSensorData.fBrightness);
END_IF
IF fBrightness_10 <> 0 THEN
	stPirSensorData.fBrightness:=  MIN(fBrightness_10, stPirSensorData.fBrightness);
END_IF


IF NOT bInitialize THEN
	FOR nIdxScan := 1 TO nNumberOfSensors DO
		fbInitTimeOut[nIdxScan](IN:= FALSE);
		arrInitDone[nIdxScan] := FALSE;
		arrInitErr[nIdxScan] := FALSE;
	END_FOR
END_IF
END_ACTION

END_FUNCTION_BLOCK

// POUs/DALI/DALI_Devices/NIKO/FB_NIKO_P46xx_1Pcs
FUNCTION_BLOCK FB_NIKO_P46xx_1Pcs
VAR_INPUT
	byShrtAdr					: BYTE;
	bInitialize					: BOOL := TRUE;
	ipCommunication				: I_DALICommunication;
	DALI_LINE_NUM				: INT := 1;	

	bCancelHoldTimerOccupancy	: BOOL;
END_VAR
VAR_OUTPUT
	bInitErr: BOOL;
	bInitDone: BOOL;
END_VAR
VAR
	fbNiko_P46xx				: FB_DALI_Niko_P46LR(0);
	
	fbDelaySetupDALIDevice		: TON;
	tDelayTime					: TIME;
	bInitSensor					: BOOL;
	fbInitDone					: F_TRIG;
	bInitializing				: BOOL;

	bQueryOccupancy				: BOOL;
	bQueryBrightness			: BOOL;



	bAutoRead					: BOOL;
	fbAutoRequestBrightness_TON	: TOF;
	bInitTimeOut				: BOOL;
	fbInitTimeOut				: Ton;
	nCheckIdx					: INT;
	bInitScalesDone				: BOOL;
END_VAR
VAR_IN_OUT
	stSensorSetup 				: ST_DALI_NIKOP46SetupData ;	
	stPirSensorData				: ST_DALI_Sensor;
	arrSensorScales				: ARRAY [1.. 10] OF ST_DALI_SensorScaleMode;
END_VAR


fbNiko_P46xx.ipDALICommunication := ipCommunication;

IF NOT bInitScalesDone THEN
	FOR nCheckIdx:= 1 TO 10 DO
		IF arrSensorScales[nCheckIdx].fMeassureMaxSensor = 0 THEN
			arrSensorScales[nCheckIdx].fMeassureMaxSensor := 1;
		END_IF
		IF arrSensorScales[nCheckIdx].fReadMaxSensor = 0 THEN
			arrSensorScales[nCheckIdx].fReadMaxSensor := 1;
		END_IF
	END_FOR
	bInitScalesDone := TRUE;
END_IF

IF ipCommunication <> 0 THEN
	A_NIKO_P46xx_1();
END_IF

ACTION A_NIKO_P46xx_1:
//Setup parameters
	//Setup Motion part of sensor (Instance 0)
	fbNiko_P46xx.bEnableOccupancy := TRUE ;
	fbNiko_P46xx.eEventPriorityOccupancy:= stSensorSetup.eEventPriorityOccupancy;
	fbNiko_P46xx.nHoldTimerOccupancy := stSensorSetup.nHoldTimerOccupancy ;
	fbNiko_P46xx.nReportTimerOccupancy := stSensorSetup.nReportTimerOccupancy;
	fbNiko_P46xx.nDeadtimeTimerOccupancy:= stSensorSetup.nDeadtimeTimerOccupancy;
	fbNiko_P46xx.nSensitivityOccupancyA:= stSensorSetup.nSensitivityPIRSegmentA;
	fbNiko_P46xx.nSensitivityOccupancyB:= stSensorSetup.nSensitivityPIRSegmentB;
	fbNiko_P46xx.nSensitivityOccupancyC:= stSensorSetup.nSensitivityPIRSegmentC;

	//Setup Brightness part of sensor (Instance 1)
	fbNiko_P46xx.bEnableBrightness := stSensorSetup.bEnableInstanceBrightness;
	fbNiko_P46xx.eEventPriorityBrightness:= stSensorSetup.eEventPriorityBrightness;
	fbNiko_P46xx.nDeadtimeTimerBrightness:= stSensorSetup.nDeadtimeTimerBrightness;
	fbNiko_P46xx.nHysteresisBrightness:= stSensorSetup.nHysteresisBrightness;
	fbNiko_P46xx.nHysteresisMinBrightness:= stSensorSetup.nHysteresisMinBrightness;
	fbNiko_P46xx.nReportTimerBrightness:= stSensorSetup.nReportTimerBrightness;
	
	
//Calculate delay time for init sensor
tDelayTime := INT_TO_TIME((BYTE_TO_INT(byShrtAdr) * 400));	
fbDelaySetupDALIDevice(IN:= bInitialize AND NOT bInitDone , PT:=tDelayTime , Q=> , ET=> );	
	
IF fbDelaySetupDALIDevice.q AND NOT GVL_DALI.arrbBlockDTR[DALI_LINE_NUM] AND NOT bInitErr THEN
	bInitDone := FALSE;
	bInitErr := FALSE;
	bInitSensor:= TRUE;
	GVL_DALI.arrbBlockDTR[DALI_LINE_NUM]:= TRUE;
END_IF

fbAutoRequestBrightness_TON(IN:= NOT fbAutoRequestBrightness_TON.Q  AND NOT stPirSensorData.bQueryBrightness , PT:= (tDelayTime + T#12M) , Q=>bAutoRead , ET=> );

bQueryBrightness:= stPirSensorData.bQueryBrightness OR NOT bAutoRead;

fbNiko_P46xx(
	bError=> , 
	ipResultMessage=> , 
	bInitialize:=  bInitSensor, 
	nShortAddress:= byShrtAdr, 
	nOptions:= , 
	bQueryOccupancy:= bQueryOccupancy, 
	bQueryBrightness:= bQueryBrightness, 
	bCancelHoldTimerOccupancy:= bCancelHoldTimerOccupancy, 
	bInitializing=> bInitializing , 
	bReadingOccupancy=> , 
	bReadingBrightness=> , 
	bOccupied=> stPirSensorData.bPrc, 
	nBrightnessLevel=> );
	
IF fbNiko_P46xx.bError THEN
	GVL_DALI_LatestError.arrLineShrtAddr[DALI_LINE_NUM] := byShrtAdr;
END_IF

fbInitDone(CLK:=bInitSensor AND bInitializing );	
	IF fbInitDone.Q THEN
		IF NOT bInitTimeOut THEN
			bInitDone := TRUE;
			bInitErr := FALSE;
			GVL_DALI.arrbBlockDTR[DALI_LINE_NUM]:= FALSE;
		ELSE
			bInitErr := TRUE;
			GVL_DALI.arrbBlockDTR[DALI_LINE_NUM]:= FALSE;
		END_IF
	END_IF


fbInitTimeOut(IN:=bInitializing, PT:= T#10S); 

IF fbInitTimeOut.Q THEN
	bInitErr := TRUE;
	GVL_DALI.arrbBlockDTR[DALI_LINE_NUM]:= FALSE;
END_IF

stPirSensorData.bBrightnessRead:= fbNiko_P46xx.bReadingBrightness ;

stPirSensorData.fBrightness:= F_fScale(0, arrSensorScales[1].fReadMaxSensor, 0, arrSensorScales[1].fMeassureMaxSensor, 0 , fbNiko_P46xx.nBrightnessLevel);
END_ACTION

END_FUNCTION_BLOCK

// POUs/DALI/DALI_Devices/NIKO/FB_NIKO_P46xx_2Pcs
FUNCTION_BLOCK FB_NIKO_P46xx_2Pcs
VAR_INPUT
	arrShrtAdr					: ARRAY [1..2] OF BYTE;
	bInitialize					: BOOL := TRUE;
	ipCommunication				: I_DALICommunication;
	DALI_LINE_NUM				: INT := 1;	
	bCancelHoldTimerOccupancy	: BOOL;

END_VAR
VAR_OUTPUT
	arrInitErr: ARRAY [1.. nNumberOfSensors] OF BOOL;
	arrInitDone: ARRAY [1.. nNumberOfSensors] OF BOOL;
END_VAR
VAR
	arrNiko_P46xx				: ARRAY [1.. nNumberOfSensors] OF FB_DALI_Niko_P46LR(0);
	
	arrDelaySetupDALIDevice		: ARRAY [1.. nNumberOfSensors] Of TON;
	arrtDelayTime				: ARRAY [1.. nNumberOfSensors] OF TIME;
	arrInitSensor				: ARRAY [1.. nNumberOfSensors] OF BOOL;
	arrInitDone_FTrig			: ARRAY [1.. nNumberOfSensors] OF F_TRIG;
	arrInitializing				: ARRAY [1.. nNumberOfSensors] OF BOOL;
	bQueryBrightness 			: BOOL;
	bQueryOccupancy				: BOOL;
//	eEventPriorityOccupancy		: E_DALIEventPriority := E_DALIEVENTPRIORITY.Middle;
//	nHoldTimerOccupancy			: WORD := 5; // Value in s. 	
//	nReportTimerOccupancy		: BYTE := 120; // Value in s, Preset manufacturer value
//	nDeadtimeTimerOccupancy		: WORD := 100; // Value in ms, Predefined Value of DALI Standard
//	nSensitivityOccupancy		: BYTE:= 3; //setting Sensivity (0..4) 0 (Off), 1 (Min), 2(Low), 3(High) and 4 (Max)
//
//	bEnableLuxEvent				: BOOL;
//	eEventPriorityBrightness	: E_DALIEventPriority := E_DALIEVENTPRIORITY.Middle;
//	nDeadtimeTimerBrightness	: WORD := 1500; // Value in ms, Predefined Value of DALI Standard
//	nHysteresisBrightness		: BYTE := 2; // Value in %
//	nHysteresisMinBrightness	: BYTE := 10; // Absolute Value, depending on the manufacturer specific resolution
//	nReportTimerBrightness		: BYTE := 120; // Value in s, Preset manufacturer value

	bAutoRead					: BOOL;
	fbAutoRequestBrightness_TON	: TOF;
	bInitTimeOut				: BOOL;
	fbInitTimeOut				: ARRAY [1.. nNumberOfSensors] OF Ton;
	nIdxScan					: BYTE;
	nPirIdxOn					: BYTE;
	bInitDone					: BOOL;
	nBrightnessIdx				: BYTE;
	bInitScalesDone				: BOOL;

	nCheckIdx					: INT;
END_VAR
VAR_IN_OUT
	stSensorSetup 				: ST_DALI_NIKOP46SetupData ;	
	stPirSensorData				: ST_DALI_Sensor;
	arrSensorScales				: ARRAY [1.. 10] OF ST_DALI_SensorScaleMode;
END_VAR

VAR CONSTANT
	nNumberOfSensors: BYTE := 2;
END_VAR


arrNiko_P46xx[1].ipDALICommunication := ipCommunication;
arrNiko_P46xx[2].ipDALICommunication := ipCommunication;

IF NOT bInitScalesDone THEN
	FOR nCheckIdx:= 1 TO 10 DO
		IF arrSensorScales[nCheckIdx].fMeassureMaxSensor = 0 THEN
			arrSensorScales[nCheckIdx].fMeassureMaxSensor := 1;
		END_IF
		IF arrSensorScales[nCheckIdx].fReadMaxSensor = 0 THEN
			arrSensorScales[nCheckIdx].fReadMaxSensor := 1;
		END_IF
	END_FOR
	bInitScalesDone := TRUE;
END_IF


IF ipCommunication <> 0 THEN
	A_NIKO_P46xx();
END_IF

ACTION A_NIKO_P46xx:


FOR nIdxScan := 1 TO nNumberOfSensors DO
	//Setup parameters
		//Setup Motion part of sensor (Instance 0)
		arrNiko_P46xx[nIdxScan].eEventPriorityOccupancy:= stSensorSetup.eEventPriorityOccupancy;
		arrNiko_P46xx[nIdxScan].nHoldTimerOccupancy := stSensorSetup.nHoldTimerOccupancy ;
		arrNiko_P46xx[nIdxScan].nReportTimerOccupancy := stSensorSetup.nReportTimerOccupancy;
		arrNiko_P46xx[nIdxScan].nDeadtimeTimerOccupancy:= stSensorSetup.nDeadtimeTimerOccupancy;
		arrNiko_P46xx[nIdxScan].nSensitivityOccupancyA:= stSensorSetup.nSensitivityPIRSegmentA;
		arrNiko_P46xx[nIdxScan].nSensitivityOccupancyB:= stSensorSetup.nSensitivityPIRSegmentB;
		arrNiko_P46xx[nIdxScan].nSensitivityOccupancyC:= stSensorSetup.nSensitivityPIRSegmentC;
	
		//Setup Brightness part of sensor (Instance 1)
		arrNiko_P46xx[nIdxScan].bEnableBrightness := stSensorSetup.bEnableInstanceBrightness;
		arrNiko_P46xx[nIdxScan].eEventPriorityBrightness:= stSensorSetup.eEventPriorityBrightness;
		arrNiko_P46xx[nIdxScan].nDeadtimeTimerBrightness:= stSensorSetup.nDeadtimeTimerBrightness;
		arrNiko_P46xx[nIdxScan].nHysteresisBrightness:= stSensorSetup.nHysteresisBrightness;
		arrNiko_P46xx[nIdxScan].nHysteresisMinBrightness:= stSensorSetup.nHysteresisMinBrightness;
		arrNiko_P46xx[nIdxScan].nReportTimerBrightness:= stSensorSetup.nReportTimerBrightness;
	
	//Calculate delay time for init sensor
	arrtDelayTime[nIdxScan] := INT_TO_TIME((BYTE_TO_INT(arrShrtAdr[nIdxScan]) * 400));	
	arrDelaySetupDALIDevice[nIdxScan](IN:= bInitialize , PT:=arrtDelayTime[nIdxScan] , Q=> , ET=> );	
		
	IF arrDelaySetupDALIDevice[nIdxScan].q AND NOT GVL_DALI.arrbBlockDTR[DALI_LINE_NUM] AND NOT (arrInitDone[nIdxScan] OR arrInitErr[nIdxScan]) THEN
		arrInitSensor[nIdxScan]:= TRUE;
		GVL_DALI.arrbBlockDTR[DALI_LINE_NUM]:= TRUE;
	END_IF
	
	bQueryBrightness:= stPirSensorData.bQueryBrightness OR NOT bAutoRead;
	
	fbAutoRequestBrightness_TON(IN:= NOT fbAutoRequestBrightness_TON.Q  AND NOT stPirSensorData.bQueryBrightness , PT:= (arrtDelayTime[nIdxScan] + T#12M) , Q=>bAutoRead , ET=> );
	
	bQueryOccupancy:= NOT bAutoRead OR stPirSensorData.bQueryBrightness;
	
	arrNiko_P46xx[nIdxScan](
		bError=> , 
		ipResultMessage=> , 
		bInitialize:=  arrInitSensor[nIdxScan], 
		nShortAddress:= arrShrtAdr[nIdxScan] , 
		nOptions:= , 
		bQueryOccupancy:= bQueryOccupancy, 
		bQueryBrightness:= bQueryBrightness, 
		bCancelHoldTimerOccupancy:= bCancelHoldTimerOccupancy, 
		bInitializing=> arrInitializing[nIdxScan] , 
		bReadingOccupancy=> , 
		bReadingBrightness=> , 
		bOccupied=> , 
		nBrightnessLevel=> );
	
	IF arrNiko_P46xx[nIdxScan].bError THEN
		GVL_DALI_LatestError.arrLineShrtAddr[DALI_LINE_NUM] := arrShrtAdr[nIdxScan];
	END_IF
	
	arrInitDone_FTrig[nIdxScan](CLK:=arrInitializing[nIdxScan] );	
		IF arrInitDone_FTrig[nIdxScan].Q THEN
			IF NOT bInitTimeOut THEN
				bInitDone := TRUE;
				GVL_DALI.arrbBlockDTR[DALI_LINE_NUM]:= FALSE;
			ELSE
				arrInitErr[nIdxScan] := TRUE;
				GVL_DALI.arrbBlockDTR[DALI_LINE_NUM]:= FALSE;
			END_IF
		END_IF
		
	fbInitTimeOut[nIdxScan](IN:=arrInitSensor[nIdxScan], PT:= T#10S); 
		IF fbInitTimeOut[nIdxScan].Q THEN
		arrInitErr[nIdxScan] := TRUE;
		GVL_DALI.arrbBlockDTR[DALI_LINE_NUM]:= FALSE;
	END_IF
END_FOR

stPirSensorData.bPrc:= FALSE;
FOR nPirIdxOn:= 1 TO nNumberOfSensors DO
	IF arrNiko_P46xx[nPirIdxOn].bOccupied THEN
		stPirSensorData.bPrc:= TRUE;
		EXIT;
	END_IF
END_FOR

stPirSensorData.bBrightnessRead:= arrNiko_P46xx[1].bReadingBrightness OR arrNiko_P46xx[2].bReadingBrightness;

stPirSensorData.fBrightness:= MIN(F_fScale(0, arrSensorScales[1].fReadMaxSensor, 0, arrSensorScales[1].fMeassureMaxSensor, 0 , arrNiko_P46xx[1].nBrightnessLevel), 
								F_fScale(0, arrSensorScales[2].fReadMaxSensor, 0, arrSensorScales[2].fMeassureMaxSensor, 0, arrNiko_P46xx[2].nBrightnessLevel));
END_ACTION

END_FUNCTION_BLOCK

// POUs/DALI/DALI_Devices/NIKO/FB_NIKO_P46xx_3Pcs
FUNCTION_BLOCK FB_NIKO_P46xx_3Pcs
VAR_INPUT
	arrShrtAdr					: ARRAY [1..3] OF BYTE;
	bInitialize					: BOOL := TRUE;
	ipCommunication				: I_DALICommunication;
	DALI_LINE_NUM				: INT := 1;	
END_VAR
VAR_OUTPUT
	bPrc 						: BOOL;
	fActualBrightness					: REAL;
	arrInitErr					: ARRAY [1.. nNumberOfSensors] OF BOOL;
	arrInitDone					: ARRAY [1.. nNumberOfSensors] OF BOOL;
END_VAR
VAR
	arrNiko_P46xx				: ARRAY [1.. nNumberOfSensors] OF FB_DALI_Niko_P46LR(0);
	
	arrDelaySetupDALIDevice		: ARRAY [1.. nNumberOfSensors] Of TON;
	arrtDelayTime				: ARRAY [1.. nNumberOfSensors] OF TIME;
	arrInitSensor				: ARRAY [1.. nNumberOfSensors] OF BOOL;
	arrInitDone_FTrig			: ARRAY [1.. nNumberOfSensors] OF F_TRIG;
	arrInitializing				: ARRAY [1.. nNumberOfSensors] OF BOOL;
	bQueryBrightness 			: BOOL;
	bQueryOccupancy				: BOOL;
	eEventPriorityOccupancy		: E_DALIEventPriority := E_DALIEVENTPRIORITY.Middle;
	nHoldTimerOccupancy			: WORD := 5; // Value in s. 	
	nReportTimerOccupancy		: BYTE := 120; // Value in s, Preset manufacturer value
	nDeadtimeTimerOccupancy		: WORD := 100; // Value in ms, Predefined Value of DALI Standard
	bCancelHoldTimerOccupancy	: BOOL;
	nSensitivityOccupancy		: BYTE:= 3; //setting Sensivity (0..4) 0 (Off), 1 (Min), 2(Low), 3(High) and 4 (Max)

	bEnableLuxEvent				: BOOL;
	eEventPriorityBrightness	: E_DALIEventPriority := E_DALIEVENTPRIORITY.Middle;
	nDeadtimeTimerBrightness	: WORD := 1500; // Value in ms, Predefined Value of DALI Standard
	nHysteresisBrightness		: BYTE := 2; // Value in %
	nHysteresisMinBrightness	: BYTE := 10; // Absolute Value, depending on the manufacturer specific resolution
	nReportTimerBrightness		: BYTE := 120; // Value in s, Preset manufacturer value

	bAutoRead					: BOOL;
	fbAutoRequestBrightness_TON	: TOF;
	bInitTimeOut				: BOOL;
	fbInitTimeOut				: ARRAY [1.. nNumberOfSensors] OF TON;
	nIdxScan					: BYTE;
	nPirIdxOn					: BYTE;
	bInitDone					: BOOL;
	bInitScalesDone				: BOOL;

	nBrightnessIdx				: BYTE;
	fBrightness_1				: REAL;
	fBrightness_2				: REAL;
	fBrightness_3				: REAL;

	nCheckIdx: INT;
END_VAR
VAR_IN_OUT
	stSensorSetup 				: ST_DALI_NIKOP46SetupData ;	
	stPirSensorData				: ST_DALI_Sensor;
	arrSensorScales				: ARRAY [1.. 10] OF ST_DALI_SensorScaleMode;
END_VAR

VAR CONSTANT
	nNumberOfSensors: BYTE := 3;
END_VAR


arrNiko_P46xx[1].ipDALICommunication := ipCommunication;
arrNiko_P46xx[2].ipDALICommunication := ipCommunication;
arrNiko_P46xx[3].ipDALICommunication := ipCommunication;

IF NOT bInitScalesDone THEN
	FOR nCheckIdx:= 1 TO 10 DO
		IF arrSensorScales[nCheckIdx].fMeassureMaxSensor = 0 THEN
			arrSensorScales[nCheckIdx].fMeassureMaxSensor := 1;
		END_IF
		IF arrSensorScales[nCheckIdx].fReadMaxSensor = 0 THEN
			arrSensorScales[nCheckIdx].fReadMaxSensor := 1;
		END_IF
	END_FOR
	bInitScalesDone := TRUE;
END_IF


IF ipCommunication <> 0 THEN
	A_NIKO_P46xx();
END_IF

ACTION A_NIKO_P46xx:


FOR nIdxScan := 1 TO nNumberOfSensors DO

	//Setup parameters
		//Setup Motion part of sensor (Instance 0)
		arrNiko_P46xx[nIdxScan].eEventPriorityOccupancy:= stSensorSetup.eEventPriorityOccupancy;
		arrNiko_P46xx[nIdxScan].nHoldTimerOccupancy := stSensorSetup.nHoldTimerOccupancy ;
		arrNiko_P46xx[nIdxScan].nReportTimerOccupancy := stSensorSetup.nReportTimerOccupancy;
		arrNiko_P46xx[nIdxScan].nDeadtimeTimerOccupancy:= stSensorSetup.nDeadtimeTimerOccupancy;
		arrNiko_P46xx[nIdxScan].nSensitivityOccupancyA:= stSensorSetup.nSensitivityPIRSegmentA;
		arrNiko_P46xx[nIdxScan].nSensitivityOccupancyB:= stSensorSetup.nSensitivityPIRSegmentB;
		arrNiko_P46xx[nIdxScan].nSensitivityOccupancyC:= stSensorSetup.nSensitivityPIRSegmentC;
	
		//Setup Brightness part of sensor (Instance 1)
		arrNiko_P46xx[nIdxScan].bEnableBrightness := stSensorSetup.bEnableInstanceBrightness;
		arrNiko_P46xx[nIdxScan].eEventPriorityBrightness:= stSensorSetup.eEventPriorityBrightness;
		arrNiko_P46xx[nIdxScan].nDeadtimeTimerBrightness:= stSensorSetup.nDeadtimeTimerBrightness;
		arrNiko_P46xx[nIdxScan].nHysteresisBrightness:= stSensorSetup.nHysteresisBrightness;
		arrNiko_P46xx[nIdxScan].nHysteresisMinBrightness:= stSensorSetup.nHysteresisMinBrightness;
		arrNiko_P46xx[nIdxScan].nReportTimerBrightness:= stSensorSetup.nReportTimerBrightness;
		
	//Calculate delay time for init sensor
	arrtDelayTime[nIdxScan] := INT_TO_TIME((BYTE_TO_INT(arrShrtAdr[nIdxScan]) * 400));	
	arrDelaySetupDALIDevice[nIdxScan](IN:= bInitialize , PT:=arrtDelayTime[nIdxScan] , Q=> , ET=> );	
		
	IF arrDelaySetupDALIDevice[nIdxScan].q AND NOT GVL_DALI.arrbBlockDTR[DALI_LINE_NUM] AND NOT (arrInitDone[nIdxScan] OR arrInitErr[nIdxScan]) THEN
		arrInitSensor[nIdxScan]:= TRUE;
		GVL_DALI.arrbBlockDTR[DALI_LINE_NUM]:= TRUE;
	END_IF
	
	bQueryBrightness:= stPirSensorData.bQueryBrightness OR NOT bAutoRead;
	
	fbAutoRequestBrightness_TON(IN:= NOT fbAutoRequestBrightness_TON.Q  AND NOT stPirSensorData.bQueryBrightness , PT:= (arrtDelayTime[nIdxScan] + T#12M) , Q=>bAutoRead , ET=> );
	
	bQueryOccupancy:= NOT bAutoRead OR stPirSensorData.bQueryBrightness;
	
	arrNiko_P46xx[nIdxScan](
		bError=> , 
		ipResultMessage=> , 
		bInitialize:=  arrInitSensor[nIdxScan], 
		nShortAddress:= arrShrtAdr[nIdxScan] , 
		nOptions:= , 
		bQueryOccupancy:= bQueryOccupancy, 
		bQueryBrightness:= bQueryBrightness, 
		bCancelHoldTimerOccupancy:= bCancelHoldTimerOccupancy, 
		bInitializing=> arrInitializing[nIdxScan] , 
		bReadingOccupancy=> , 
		bReadingBrightness=> , 
		bOccupied=> , 
		nBrightnessLevel=> );
	
	IF arrNiko_P46xx[nIdxScan].bError THEN
		GVL_DALI_LatestError.arrLineShrtAddr[DALI_LINE_NUM] := arrShrtAdr[nIdxScan];
	END_IF
	
	arrInitDone_FTrig[nIdxScan](CLK:=arrInitializing[nIdxScan] );	
		IF arrInitDone_FTrig[nIdxScan].Q THEN
			IF NOT bInitTimeOut THEN
				arrInitDone[nIdxScan] := TRUE;
				GVL_DALI.arrbBlockDTR[DALI_LINE_NUM]:= FALSE;
			ELSE
				arrInitErr[nIdxScan] := TRUE;
				GVL_DALI.arrbBlockDTR[DALI_LINE_NUM]:= FALSE;
			END_IF
		END_IF
		
	fbInitTimeOut[nIdxScan](IN:=arrInitSensor[nIdxScan] AND NOT arrInitDone[nIdxScan], PT:= T#10S); 
	
	IF fbInitTimeOut[nIdxScan].Q THEN
		arrInitErr[nIdxScan] := TRUE;
		GVL_DALI.arrbBlockDTR[DALI_LINE_NUM]:= FALSE;
	END_IF
END_FOR

stPirSensorData.bPrc:= FALSE;
FOR nPirIdxOn:= 1 TO nNumberOfSensors DO
	IF arrNiko_P46xx[nPirIdxOn].bOccupied THEN
		stPirSensorData.bPrc:= TRUE;
		EXIT;
	END_IF
END_FOR
bPrc := stPirSensorData.bPrc;

stPirSensorData.bBrightnessRead:= arrNiko_P46xx[1].bReadingBrightness OR arrNiko_P46xx[2].bReadingBrightness OR arrNiko_P46xx[3].bReadingBrightness;



fBrightness_1:= F_fScale(0, arrSensorScales[1].fReadMaxSensor, 0, arrSensorScales[1].fMeassureMaxSensor, 0, arrNiko_P46xx[1].nBrightnessLevel);
fBrightness_2:= F_fScale(0, arrSensorScales[2].fReadMaxSensor, 0, arrSensorScales[2].fMeassureMaxSensor, 0, arrNiko_P46xx[2].nBrightnessLevel);
fBrightness_3:= F_fScale(0, arrSensorScales[3].fReadMaxSensor, 0, arrSensorScales[3].fMeassureMaxSensor, 0, arrNiko_P46xx[3].nBrightnessLevel);


IF fBrightness_1 <> 0 THEN
	stPirSensorData.fBrightness:= fBrightness_1;
END_IF
IF fBrightness_2 <> 0 THEN
	stPirSensorData.fBrightness:= MIN(fBrightness_2, stPirSensorData.fBrightness);
END_IF
IF fBrightness_3 <> 0 THEN
	stPirSensorData.fBrightness:=  MIN(fBrightness_3, stPirSensorData.fBrightness);
END_IF

fActualBrightness := stPirSensorData.fBrightness ;

IF NOT bInitialize THEN
	FOR nIdxScan := 1 TO nNumberOfSensors DO
		fbInitTimeOut[nIdxScan](IN:= FALSE);
		arrInitDone[nIdxScan] := FALSE;
		arrInitErr[nIdxScan] := FALSE;
	END_FOR
END_IF
END_ACTION

END_FUNCTION_BLOCK

// POUs/DALI/DALI_Devices/NIKO/FB_NIKO_P46xx_4Pcs
FUNCTION_BLOCK FB_NIKO_P46xx_4Pcs
VAR_INPUT
	arrShrtAdr					: ARRAY [1..4] OF BYTE;
	bInitialize					: BOOL := TRUE;
	ipCommunication				: I_DALICommunication;
	DALI_LINE_NUM				: INT := 1;	

END_VAR
VAR_OUTPUT
	arrInitErr: ARRAY [1.. nNumberOfSensors] OF BOOL;
	arrInitDone: ARRAY [1.. nNumberOfSensors] OF BOOL;
END_VAR
VAR
	arrNiko_P46xx				: ARRAY [1.. nNumberOfSensors] OF FB_DALI_Niko_P46LR(0);
	
	arrDelaySetupDALIDevice		: ARRAY [1.. nNumberOfSensors] Of TON;
	arrtDelayTime				: ARRAY [1.. nNumberOfSensors] OF TIME;
	arrInitSensor				: ARRAY [1.. nNumberOfSensors] OF BOOL;
	arrInitDone_FTrig			: ARRAY [1.. nNumberOfSensors] OF F_TRIG;
	arrInitializing				: ARRAY [1.. nNumberOfSensors] OF BOOL;
	bQueryBrightness 			: BOOL;
	bQueryOccupancy				: BOOL;
	eEventPriorityOccupancy		: E_DALIEventPriority := E_DALIEVENTPRIORITY.Middle;
	nHoldTimerOccupancy			: WORD := 5; // Value in s. 	
	nReportTimerOccupancy		: BYTE := 120; // Value in s, Preset manufacturer value
	nDeadtimeTimerOccupancy		: WORD := 100; // Value in ms, Predefined Value of DALI Standard
	bCancelHoldTimerOccupancy	: BOOL;
	nSensitivityOccupancy		: BYTE:= 3; //setting Sensivity (0..4) 0 (Off), 1 (Min), 2(Low), 3(High) and 4 (Max)

	bEnableLuxEvent				: BOOL;
	eEventPriorityBrightness	: E_DALIEventPriority := E_DALIEVENTPRIORITY.Middle;
	nDeadtimeTimerBrightness	: WORD := 1500; // Value in ms, Predefined Value of DALI Standard
	nHysteresisBrightness		: BYTE := 2; // Value in %
	nHysteresisMinBrightness	: BYTE := 10; // Absolute Value, depending on the manufacturer specific resolution
	nReportTimerBrightness		: BYTE := 120; // Value in s, Preset manufacturer value

	bAutoRead					: BOOL;
	fbAutoRequestBrightness_TON	: TOF;
	bInitTimeOut				: BOOL;
	fbInitTimeOut				: ARRAY [1.. nNumberOfSensors] OF TON;
	nIdxScan					: BYTE;
	nPirIdxOn					: BYTE;
	bInitDone					: BOOL;
	nBrightnessIdx				: BYTE;
	bInitScalesDone				: BOOL;
	fBrightness_1				: REAL;
	fBrightness_2				: REAL;
	fBrightness_3				: REAL;
	fBrightness_4				: REAL;

	nCheckIdx: INT;
END_VAR
VAR_IN_OUT
	stSensorSetup 				: ST_DALI_NIKOP46SetupData ;	
	stPirSensorData				: ST_DALI_Sensor;
	arrSensorScales				: ARRAY [1.. 10] OF ST_DALI_SensorScaleMode;
END_VAR

VAR CONSTANT
	nNumberOfSensors: BYTE := 4;
END_VAR


arrNiko_P46xx[1].ipDALICommunication := ipCommunication;
arrNiko_P46xx[2].ipDALICommunication := ipCommunication;
arrNiko_P46xx[3].ipDALICommunication := ipCommunication;
arrNiko_P46xx[4].ipDALICommunication := ipCommunication;

IF NOT bInitScalesDone THEN
	FOR nCheckIdx:= 1 TO 10 DO
		IF arrSensorScales[nCheckIdx].fMeassureMaxSensor = 0 THEN
			arrSensorScales[nCheckIdx].fMeassureMaxSensor := 1;
		END_IF
		IF arrSensorScales[nCheckIdx].fReadMaxSensor = 0 THEN
			arrSensorScales[nCheckIdx].fReadMaxSensor := 1;
		END_IF
	END_FOR
	bInitScalesDone := TRUE;
END_IF


IF ipCommunication <> 0 THEN
	A_NIKO_P46xx();
END_IF

ACTION A_NIKO_P46xx:


FOR nIdxScan := 1 TO nNumberOfSensors DO
	//Setup parameters
		//Setup Motion part of sensor (Instance 0)
		arrNiko_P46xx[nIdxScan].eEventPriorityOccupancy:= stSensorSetup.eEventPriorityOccupancy;
		arrNiko_P46xx[nIdxScan].nHoldTimerOccupancy := stSensorSetup.nHoldTimerOccupancy ;
		arrNiko_P46xx[nIdxScan].nReportTimerOccupancy := stSensorSetup.nReportTimerOccupancy;
		arrNiko_P46xx[nIdxScan].nDeadtimeTimerOccupancy:= stSensorSetup.nDeadtimeTimerOccupancy;
		arrNiko_P46xx[nIdxScan].nSensitivityOccupancyA:= stSensorSetup.nSensitivityPIRSegmentA;
		arrNiko_P46xx[nIdxScan].nSensitivityOccupancyB:= stSensorSetup.nSensitivityPIRSegmentB;
		arrNiko_P46xx[nIdxScan].nSensitivityOccupancyC:= stSensorSetup.nSensitivityPIRSegmentC;
	
		//Setup Brightness part of sensor (Instance 1)
		arrNiko_P46xx[nIdxScan].bEnableBrightness := stSensorSetup.bEnableInstanceBrightness;
		arrNiko_P46xx[nIdxScan].eEventPriorityBrightness:= stSensorSetup.eEventPriorityBrightness;
		arrNiko_P46xx[nIdxScan].nDeadtimeTimerBrightness:= stSensorSetup.nDeadtimeTimerBrightness;
		arrNiko_P46xx[nIdxScan].nHysteresisBrightness:= stSensorSetup.nHysteresisBrightness;
		arrNiko_P46xx[nIdxScan].nHysteresisMinBrightness:= stSensorSetup.nHysteresisMinBrightness;
		arrNiko_P46xx[nIdxScan].nReportTimerBrightness:= stSensorSetup.nReportTimerBrightness;
		
	
	//Calculate delay time for init sensor
	arrtDelayTime[nIdxScan] := INT_TO_TIME((BYTE_TO_INT(arrShrtAdr[nIdxScan]) * 400));	
	arrDelaySetupDALIDevice[nIdxScan](IN:= bInitialize , PT:=arrtDelayTime[nIdxScan] , Q=> , ET=> );	
		
	IF arrDelaySetupDALIDevice[nIdxScan].q AND NOT GVL_DALI.arrbBlockDTR[DALI_LINE_NUM] AND NOT (arrInitDone[nIdxScan] OR arrInitErr[nIdxScan]) THEN
		arrInitSensor[nIdxScan]:= TRUE;
		GVL_DALI.arrbBlockDTR[DALI_LINE_NUM]:= TRUE;
	END_IF
	
	bQueryBrightness:= stPirSensorData.bQueryBrightness OR NOT bAutoRead;
	
	fbAutoRequestBrightness_TON(IN:= NOT fbAutoRequestBrightness_TON.Q  AND NOT stPirSensorData.bQueryBrightness , PT:= (arrtDelayTime[nIdxScan] + T#12M) , Q=>bAutoRead , ET=> );
	
	bQueryOccupancy:= NOT bAutoRead OR stPirSensorData.bQueryBrightness;
	
	arrNiko_P46xx[nIdxScan](
		bError=> , 
		ipResultMessage=> , 
		bInitialize:=  arrInitSensor[nIdxScan], 
		nShortAddress:= arrShrtAdr[nIdxScan], 
		nOptions:= , 
		bQueryOccupancy:= bQueryOccupancy, 
		bQueryBrightness:= bQueryBrightness, 
		bCancelHoldTimerOccupancy:= bCancelHoldTimerOccupancy, 
		bInitializing=> arrInitializing[nIdxScan] , 
		bReadingOccupancy=> , 
		bReadingBrightness=> , 
		bOccupied=> , 
		nBrightnessLevel=> );
	
	IF arrNiko_P46xx[nIdxScan].bError THEN
		GVL_DALI_LatestError.arrLineShrtAddr[DALI_LINE_NUM] := arrShrtAdr[nIdxScan];
	END_IF
	
	arrInitDone_FTrig[nIdxScan](CLK:=arrInitializing[nIdxScan] );	
		IF arrInitDone_FTrig[nIdxScan].Q THEN
			IF NOT bInitTimeOut THEN
				arrInitDone[nIdxScan] := TRUE;
				GVL_DALI.arrbBlockDTR[DALI_LINE_NUM]:= FALSE;
			ELSE
				arrInitErr[nIdxScan] := TRUE;
				GVL_DALI.arrbBlockDTR[DALI_LINE_NUM]:= FALSE;
			END_IF
		END_IF
		
	fbInitTimeOut[nIdxScan](IN:=arrInitSensor[nIdxScan] AND NOT arrInitDone[nIdxScan], PT:= T#10S); 
	
	IF fbInitTimeOut[nIdxScan].Q THEN
		arrInitErr[nIdxScan] := TRUE;
		GVL_DALI.arrbBlockDTR[DALI_LINE_NUM]:= FALSE;
	END_IF
END_FOR

stPirSensorData.bPrc:= FALSE;
FOR nPirIdxOn:= 1 TO nNumberOfSensors DO
	IF arrNiko_P46xx[nPirIdxOn].bOccupied THEN
		stPirSensorData.bPrc:= TRUE;
		EXIT;
	END_IF
END_FOR

stPirSensorData.bBrightnessRead:= arrNiko_P46xx[1].bReadingBrightness OR arrNiko_P46xx[2].bReadingBrightness OR arrNiko_P46xx[3].bReadingBrightness OR arrNiko_P46xx[4].bReadingBrightness;



fBrightness_1:= F_fScale(0, arrSensorScales[1].fReadMaxSensor, 0, arrSensorScales[1].fMeassureMaxSensor, 0, arrNiko_P46xx[1].nBrightnessLevel);
fBrightness_2:= F_fScale(0, arrSensorScales[2].fReadMaxSensor, 0, arrSensorScales[2].fMeassureMaxSensor, 0, arrNiko_P46xx[2].nBrightnessLevel);
fBrightness_3:= F_fScale(0, arrSensorScales[3].fReadMaxSensor, 0, arrSensorScales[3].fMeassureMaxSensor, 0, arrNiko_P46xx[3].nBrightnessLevel);
fBrightness_4:= F_fScale(0, arrSensorScales[4].fReadMaxSensor, 0, arrSensorScales[4].fMeassureMaxSensor, 0, arrNiko_P46xx[4].nBrightnessLevel);


IF fBrightness_1 <> 0 THEN
	stPirSensorData.fBrightness:= fBrightness_1;
ELSE
	stPirSensorData.fBrightness:= 9999;
END_IF
IF fBrightness_2 <> 0 THEN
	stPirSensorData.fBrightness:= MIN(fBrightness_2, stPirSensorData.fBrightness);
END_IF
IF fBrightness_3 <> 0 THEN
	stPirSensorData.fBrightness:=  MIN(fBrightness_3, stPirSensorData.fBrightness);
END_IF
IF fBrightness_4 <> 0 THEN
	stPirSensorData.fBrightness:=  MIN(fBrightness_4, stPirSensorData.fBrightness);
END_IF

IF NOT bInitialize THEN
	FOR nIdxScan := 1 TO nNumberOfSensors DO
		fbInitTimeOut[nIdxScan](IN:= FALSE);
		arrInitDone[nIdxScan] := FALSE;
		arrInitErr[nIdxScan] := FALSE;
	END_FOR
END_IF
END_ACTION

END_FUNCTION_BLOCK

// POUs/DALI/DALI_Devices/NIKO/FB_NIKO_P46xx_5Pcs
FUNCTION_BLOCK FB_NIKO_P46xx_5Pcs
VAR_INPUT
	arrShrtAdr					: ARRAY [1..5] OF BYTE;
	bInitialize					: BOOL := TRUE;
	ipCommunication				: I_DALICommunication;
	DALI_LINE_NUM				: INT := 1;	
END_VAR
VAR_OUTPUT
	arrInitErr: ARRAY [1.. nNumberOfSensors] OF BOOL;
	arrInitDone: ARRAY [1.. nNumberOfSensors] OF BOOL;
END_VAR
VAR
	arrNiko_P46xx				: ARRAY [1.. nNumberOfSensors] OF FB_DALI_Niko_P46LR(0);
	
	arrDelaySetupDALIDevice		: ARRAY [1.. nNumberOfSensors] Of TON;
	arrtDelayTime				: ARRAY [1.. nNumberOfSensors] OF TIME;
	arrInitSensor				: ARRAY [1.. nNumberOfSensors] OF BOOL;
	arrInitDone_FTrig			: ARRAY [1.. nNumberOfSensors] OF F_TRIG;
	arrInitializing				: ARRAY [1.. nNumberOfSensors] OF BOOL;
	bQueryBrightness 			: BOOL;
	bQueryOccupancy				: BOOL;
	eEventPriorityOccupancy		: E_DALIEventPriority := E_DALIEVENTPRIORITY.Middle;
	nHoldTimerOccupancy			: WORD := 5; // Value in s. 	
	nReportTimerOccupancy		: BYTE := 120; // Value in s, Preset manufacturer value
	nDeadtimeTimerOccupancy		: WORD := 100; // Value in ms, Predefined Value of DALI Standard
	bCancelHoldTimerOccupancy	: BOOL;
	nSensitivityOccupancy		: BYTE:= 3; //setting Sensivity (0..4) 0 (Off), 1 (Min), 2(Low), 3(High) and 4 (Max)

	bEnableLuxEvent				: BOOL;
	eEventPriorityBrightness	: E_DALIEventPriority := E_DALIEVENTPRIORITY.Middle;
	nDeadtimeTimerBrightness	: WORD := 1500; // Value in ms, Predefined Value of DALI Standard
	nHysteresisBrightness		: BYTE := 2; // Value in %
	nHysteresisMinBrightness	: BYTE := 10; // Absolute Value, depending on the manufacturer specific resolution
	nReportTimerBrightness		: BYTE := 120; // Value in s, Preset manufacturer value

	bAutoRead					: BOOL;
	fbAutoRequestBrightness_TON	: TOF;
	bInitTimeOut				: BOOL;
	fbInitTimeOut				: ARRAY [1.. nNumberOfSensors] OF TON;
	nIdxScan					: BYTE;
	nPirIdxOn					: BYTE;
	nBrightnessIdx				: BYTE;
	fBrightness_1				: REAL;
	fBrightness_2				: REAL;
	fBrightness_3				: REAL;
	fBrightness_4				: REAL;
	fBrightness_5				: REAL;
	bInitDone					: BOOL;
	bInitScalesDone				: BOOL;
	
	nCheckIdx: INT;
END_VAR
VAR_IN_OUT
	stSensorSetup 				: ST_DALI_NIKOP46SetupData ;	
	stPirSensorData				: ST_DALI_Sensor;
	arrSensorScales				: ARRAY [1.. 10] OF ST_DALI_SensorScaleMode;
END_VAR

VAR CONSTANT
	nNumberOfSensors: BYTE := 5;
END_VAR


arrNiko_P46xx[1].ipDALICommunication := ipCommunication;
arrNiko_P46xx[2].ipDALICommunication := ipCommunication;
arrNiko_P46xx[3].ipDALICommunication := ipCommunication;
arrNiko_P46xx[4].ipDALICommunication := ipCommunication;
arrNiko_P46xx[5].ipDALICommunication := ipCommunication;

IF NOT bInitScalesDone THEN
	FOR nCheckIdx:= 1 TO 10 DO
		IF arrSensorScales[nCheckIdx].fMeassureMaxSensor = 0 THEN
			arrSensorScales[nCheckIdx].fMeassureMaxSensor := 1;
		END_IF
		IF arrSensorScales[nCheckIdx].fReadMaxSensor = 0 THEN
			arrSensorScales[nCheckIdx].fReadMaxSensor := 1;
		END_IF
	END_FOR
	bInitScalesDone := TRUE;
END_IF

IF ipCommunication <> 0 THEN
	A_NIKO_P46xx();
END_IF

ACTION A_NIKO_P46xx:


FOR nIdxScan := 1 TO nNumberOfSensors DO
	//Setup parameters
		//Setup Motion part of sensor (Instance 0)
		arrNiko_P46xx[nIdxScan].eEventPriorityOccupancy:= stSensorSetup.eEventPriorityOccupancy;
		arrNiko_P46xx[nIdxScan].nHoldTimerOccupancy := stSensorSetup.nHoldTimerOccupancy ;
		arrNiko_P46xx[nIdxScan].nReportTimerOccupancy := stSensorSetup.nReportTimerOccupancy;
		arrNiko_P46xx[nIdxScan].nDeadtimeTimerOccupancy:= stSensorSetup.nDeadtimeTimerOccupancy;
		arrNiko_P46xx[nIdxScan].nSensitivityOccupancyA:= stSensorSetup.nSensitivityPIRSegmentA;
		arrNiko_P46xx[nIdxScan].nSensitivityOccupancyB:= stSensorSetup.nSensitivityPIRSegmentB;
		arrNiko_P46xx[nIdxScan].nSensitivityOccupancyC:= stSensorSetup.nSensitivityPIRSegmentC;
	
		//Setup Brightness part of sensor (Instance 1)
		arrNiko_P46xx[nIdxScan].bEnableBrightness := stSensorSetup.bEnableInstanceBrightness;
		arrNiko_P46xx[nIdxScan].eEventPriorityBrightness:= stSensorSetup.eEventPriorityBrightness;
		arrNiko_P46xx[nIdxScan].nDeadtimeTimerBrightness:= stSensorSetup.nDeadtimeTimerBrightness;
		arrNiko_P46xx[nIdxScan].nHysteresisBrightness:= stSensorSetup.nHysteresisBrightness;
		arrNiko_P46xx[nIdxScan].nHysteresisMinBrightness:= stSensorSetup.nHysteresisMinBrightness;
		arrNiko_P46xx[nIdxScan].nReportTimerBrightness:= stSensorSetup.nReportTimerBrightness;
		
	//Calculate delay time for init sensor
	arrtDelayTime[nIdxScan] := INT_TO_TIME((BYTE_TO_INT(arrShrtAdr[nIdxScan]) * 400));	
	arrDelaySetupDALIDevice[nIdxScan](IN:= bInitialize , PT:=arrtDelayTime[nIdxScan] , Q=> , ET=> );	
		
	IF arrDelaySetupDALIDevice[nIdxScan].q AND NOT GVL_DALI.arrbBlockDTR[DALI_LINE_NUM] AND NOT (arrInitDone[nIdxScan] OR arrInitErr[nIdxScan]) THEN
		arrInitSensor[nIdxScan]:= TRUE;
		GVL_DALI.arrbBlockDTR[DALI_LINE_NUM]:= TRUE;
	END_IF
	
	bQueryBrightness:= stPirSensorData.bQueryBrightness OR NOT bAutoRead;
	
	fbAutoRequestBrightness_TON(IN:= NOT fbAutoRequestBrightness_TON.Q  AND NOT stPirSensorData.bQueryBrightness , PT:= (arrtDelayTime[nIdxScan] + T#12M) , Q=>bAutoRead , ET=> );
	
	bQueryOccupancy:= NOT bAutoRead OR stPirSensorData.bQueryBrightness;
	
	arrNiko_P46xx[nIdxScan](
		bError=> , 
		ipResultMessage=> , 
		bInitialize:=  arrInitSensor[nIdxScan], 
		nShortAddress:= arrShrtAdr[nIdxScan], 
		nOptions:= , 
		bQueryOccupancy:= bQueryOccupancy, 
		bQueryBrightness:= bQueryBrightness, 
		bCancelHoldTimerOccupancy:= bCancelHoldTimerOccupancy, 
		bInitializing=> arrInitializing[nIdxScan] , 
		bReadingOccupancy=> , 
		bReadingBrightness=> , 
		bOccupied=> , 
		nBrightnessLevel=> );
	
	IF arrNiko_P46xx[nIdxScan].bError THEN
		GVL_DALI_LatestError.arrLineShrtAddr[DALI_LINE_NUM] :=arrShrtAdr[nIdxScan];
	END_IF
	
	arrInitDone_FTrig[nIdxScan](CLK:=arrInitializing[nIdxScan] );	
		IF arrInitDone_FTrig[nIdxScan].Q THEN
			IF NOT bInitTimeOut THEN
				arrInitDone[nIdxScan] := TRUE;
				GVL_DALI.arrbBlockDTR[DALI_LINE_NUM]:= FALSE;
			ELSE
				arrInitErr[nIdxScan] := TRUE;
				GVL_DALI.arrbBlockDTR[DALI_LINE_NUM]:= FALSE;
			END_IF
		END_IF
		
	fbInitTimeOut[nIdxScan](IN:=arrInitSensor[nIdxScan] AND NOT arrInitDone[nIdxScan], PT:= T#10S); 
	
	IF fbInitTimeOut[nIdxScan].Q THEN
		arrInitErr[nIdxScan] := TRUE;
		GVL_DALI.arrbBlockDTR[DALI_LINE_NUM]:= FALSE;
	END_IF
END_FOR

stPirSensorData.bPrc:= FALSE;
FOR nPirIdxOn:= 1 TO nNumberOfSensors DO
	IF arrNiko_P46xx[nPirIdxOn].bOccupied THEN
		stPirSensorData.bPrc:= TRUE;
		EXIT;
	END_IF
END_FOR

stPirSensorData.bBrightnessRead:= arrNiko_P46xx[1].bReadingBrightness OR arrNiko_P46xx[2].bReadingBrightness OR arrNiko_P46xx[3].bReadingBrightness OR arrNiko_P46xx[4].bReadingBrightness OR arrNiko_P46xx[5].bReadingBrightness;

fBrightness_1:= F_fScale(0, arrSensorScales[1].fReadMaxSensor, 0, arrSensorScales[1].fMeassureMaxSensor, 0, arrNiko_P46xx[1].nBrightnessLevel);
fBrightness_2:= F_fScale(0, arrSensorScales[2].fReadMaxSensor, 0, arrSensorScales[2].fMeassureMaxSensor, 0, arrNiko_P46xx[2].nBrightnessLevel);
fBrightness_3:= F_fScale(0, arrSensorScales[3].fReadMaxSensor, 0, arrSensorScales[3].fMeassureMaxSensor, 0, arrNiko_P46xx[3].nBrightnessLevel);
fBrightness_4:= F_fScale(0, arrSensorScales[4].fReadMaxSensor, 0, arrSensorScales[4].fMeassureMaxSensor, 0, arrNiko_P46xx[4].nBrightnessLevel);
fBrightness_5:= F_fScale(0, arrSensorScales[5].fReadMaxSensor, 0, arrSensorScales[5].fMeassureMaxSensor, 0, arrNiko_P46xx[5].nBrightnessLevel);


IF fBrightness_1 <> 0 THEN
	stPirSensorData.fBrightness:= fBrightness_1;
END_IF
IF fBrightness_2 <> 0 THEN
	stPirSensorData.fBrightness:= MIN(fBrightness_2, stPirSensorData.fBrightness);
END_IF
IF fBrightness_3 <> 0 THEN
	stPirSensorData.fBrightness:=  MIN(fBrightness_3, stPirSensorData.fBrightness);
END_IF
IF fBrightness_4 <> 0 THEN
	stPirSensorData.fBrightness:=  MIN(fBrightness_4, stPirSensorData.fBrightness);
END_IF
IF fBrightness_5 <> 0 THEN
	stPirSensorData.fBrightness:=  MIN(fBrightness_5, stPirSensorData.fBrightness);
END_IF


IF NOT bInitialize THEN
	FOR nIdxScan := 1 TO nNumberOfSensors DO
		fbInitTimeOut[nIdxScan](IN:= FALSE);
		arrInitDone[nIdxScan] := FALSE;
		arrInitErr[nIdxScan] := FALSE;
	END_FOR
END_IF
END_ACTION

END_FUNCTION_BLOCK

// POUs/DALI/DALI_Devices/NIKO/FB_NIKO_P46xx_6Pcs
FUNCTION_BLOCK FB_NIKO_P46xx_6Pcs
VAR_INPUT
	arrShrtAdr					: ARRAY [1..6] OF BYTE;
	bInitialize					: BOOL := TRUE;
	ipCommunication				: I_DALICommunication;
	DALI_LINE_NUM				: INT := 1;	
END_VAR
VAR_OUTPUT
	arrInitErr: ARRAY [1.. nNumberOfSensors] OF BOOL;
	arrInitDone: ARRAY [1.. nNumberOfSensors] OF BOOL;
END_VAR
VAR
	arrNiko_P46xx				: ARRAY [1.. nNumberOfSensors] OF FB_DALI_Niko_P46LR(0);
	
	arrDelaySetupDALIDevice		: ARRAY [1.. nNumberOfSensors] Of TON;
	arrtDelayTime				: ARRAY [1.. nNumberOfSensors] OF TIME;
	arrInitSensor				: ARRAY [1.. nNumberOfSensors] OF BOOL;
	arrInitDone_FTrig			: ARRAY [1.. nNumberOfSensors] OF F_TRIG;
	arrInitializing				: ARRAY [1.. nNumberOfSensors] OF BOOL;
	bQueryBrightness 			: BOOL;
	bQueryOccupancy				: BOOL;
	eEventPriorityOccupancy		: E_DALIEventPriority := E_DALIEVENTPRIORITY.Middle;
	nHoldTimerOccupancy			: WORD := 5; // Value in s. 	
	nReportTimerOccupancy		: BYTE := 120; // Value in s, Preset manufacturer value
	nDeadtimeTimerOccupancy		: WORD := 100; // Value in ms, Predefined Value of DALI Standard
	bCancelHoldTimerOccupancy	: BOOL;
	nSensitivityOccupancy		: BYTE:= 3; //setting Sensivity (0..4) 0 (Off), 1 (Min), 2(Low), 3(High) and 4 (Max)

	bEnableLuxEvent				: BOOL;
	eEventPriorityBrightness	: E_DALIEventPriority := E_DALIEVENTPRIORITY.Middle;
	nDeadtimeTimerBrightness	: WORD := 1500; // Value in ms, Predefined Value of DALI Standard
	nHysteresisBrightness		: BYTE := 2; // Value in %
	nHysteresisMinBrightness	: BYTE := 10; // Absolute Value, depending on the manufacturer specific resolution
	nReportTimerBrightness		: BYTE := 120; // Value in s, Preset manufacturer value

	bAutoRead					: BOOL;
	fbAutoRequestBrightness_TON	: TOF;
	bInitTimeOut				: BOOL;
	fbInitTimeOut				: ARRAY [1.. nNumberOfSensors] OF TON;
	nIdxScan					: BYTE;
	nPirIdxOn					: BYTE;
	nBrightnessIdx				: BYTE;
	fBrightness_1				: REAL;
	fBrightness_2				: REAL;
	fBrightness_3				: REAL;
	fBrightness_4				: REAL;
	fBrightness_5				: REAL;
	fBrightness_6				: REAL;
	bInitDone					: BOOL;
	bInitScalesDone				: BOOL;
	
	nCheckIdx: INT;
END_VAR
VAR_IN_OUT
	stSensorSetup 				: ST_DALI_NIKOP46SetupData ;	
	stPirSensorData				: ST_DALI_Sensor;
	arrSensorScales				: ARRAY [1.. 10] OF ST_DALI_SensorScaleMode;
END_VAR

VAR CONSTANT
	nNumberOfSensors: BYTE := 6;
END_VAR


arrNiko_P46xx[1].ipDALICommunication := ipCommunication;
arrNiko_P46xx[2].ipDALICommunication := ipCommunication;
arrNiko_P46xx[3].ipDALICommunication := ipCommunication;
arrNiko_P46xx[4].ipDALICommunication := ipCommunication;
arrNiko_P46xx[5].ipDALICommunication := ipCommunication;
arrNiko_P46xx[6].ipDALICommunication := ipCommunication;

IF NOT bInitScalesDone THEN
	FOR nCheckIdx:= 1 TO 10 DO
		IF arrSensorScales[nCheckIdx].fMeassureMaxSensor = 0 THEN
			arrSensorScales[nCheckIdx].fMeassureMaxSensor := 1;
		END_IF
		IF arrSensorScales[nCheckIdx].fReadMaxSensor = 0 THEN
			arrSensorScales[nCheckIdx].fReadMaxSensor := 1;
		END_IF
	END_FOR
	bInitScalesDone := TRUE;
END_IF

IF ipCommunication <> 0 THEN
	A_NIKO_P46xx();
END_IF

ACTION A_NIKO_P46xx:


FOR nIdxScan := 1 TO nNumberOfSensors DO
	//Setup parameters
		//Setup Motion part of sensor (Instance 0)
		arrNiko_P46xx[nIdxScan].eEventPriorityOccupancy:= stSensorSetup.eEventPriorityOccupancy;
		arrNiko_P46xx[nIdxScan].nHoldTimerOccupancy := stSensorSetup.nHoldTimerOccupancy ;
		arrNiko_P46xx[nIdxScan].nReportTimerOccupancy := stSensorSetup.nReportTimerOccupancy;
		arrNiko_P46xx[nIdxScan].nDeadtimeTimerOccupancy:= stSensorSetup.nDeadtimeTimerOccupancy;
		arrNiko_P46xx[nIdxScan].nSensitivityOccupancyA:= stSensorSetup.nSensitivityPIRSegmentA;
		arrNiko_P46xx[nIdxScan].nSensitivityOccupancyB:= stSensorSetup.nSensitivityPIRSegmentB;
		arrNiko_P46xx[nIdxScan].nSensitivityOccupancyC:= stSensorSetup.nSensitivityPIRSegmentC;
	
		//Setup Brightness part of sensor (Instance 1)
		arrNiko_P46xx[nIdxScan].bEnableBrightness := stSensorSetup.bEnableInstanceBrightness;
		arrNiko_P46xx[nIdxScan].eEventPriorityBrightness:= stSensorSetup.eEventPriorityBrightness;
		arrNiko_P46xx[nIdxScan].nDeadtimeTimerBrightness:= stSensorSetup.nDeadtimeTimerBrightness;
		arrNiko_P46xx[nIdxScan].nHysteresisBrightness:= stSensorSetup.nHysteresisBrightness;
		arrNiko_P46xx[nIdxScan].nHysteresisMinBrightness:= stSensorSetup.nHysteresisMinBrightness;
		arrNiko_P46xx[nIdxScan].nReportTimerBrightness:= stSensorSetup.nReportTimerBrightness;
		
	//Calculate delay time for init sensor
	arrtDelayTime[nIdxScan] := INT_TO_TIME((BYTE_TO_INT(arrShrtAdr[nIdxScan]) * 400));	
	arrDelaySetupDALIDevice[nIdxScan](IN:= bInitialize , PT:=arrtDelayTime[nIdxScan] , Q=> , ET=> );	
		
	IF arrDelaySetupDALIDevice[nIdxScan].q AND NOT GVL_DALI.arrbBlockDTR[DALI_LINE_NUM] AND NOT (arrInitDone[nIdxScan] OR arrInitErr[nIdxScan]) THEN
		arrInitSensor[nIdxScan]:= TRUE;
		GVL_DALI.arrbBlockDTR[DALI_LINE_NUM]:= TRUE;
	END_IF
	
	bQueryBrightness:= stPirSensorData.bQueryBrightness OR NOT bAutoRead;
	
	fbAutoRequestBrightness_TON(IN:= NOT fbAutoRequestBrightness_TON.Q  AND NOT stPirSensorData.bQueryBrightness , PT:= (arrtDelayTime[nIdxScan] + T#12M) , Q=>bAutoRead , ET=> );
	
	bQueryOccupancy:= NOT bAutoRead OR stPirSensorData.bQueryBrightness;
	
	arrNiko_P46xx[nIdxScan](
		bError=> , 
		ipResultMessage=> , 
		bInitialize:=  arrInitSensor[nIdxScan], 
		nShortAddress:= arrShrtAdr[nIdxScan], 
		nOptions:= , 
		bQueryOccupancy:= bQueryOccupancy, 
		bQueryBrightness:= bQueryBrightness, 
		bCancelHoldTimerOccupancy:= bCancelHoldTimerOccupancy, 
		bInitializing=> arrInitializing[nIdxScan] , 
		bReadingOccupancy=> , 
		bReadingBrightness=> , 
		bOccupied=> , 
		nBrightnessLevel=> );
	
	IF arrNiko_P46xx[nIdxScan].bError THEN
		GVL_DALI_LatestError.arrLineShrtAddr[DALI_LINE_NUM] := arrShrtAdr[nIdxScan];
	END_IF
	
	arrInitDone_FTrig[nIdxScan](CLK:=arrInitializing[nIdxScan] );	
		IF arrInitDone_FTrig[nIdxScan].Q THEN
			IF NOT bInitTimeOut THEN
				arrInitDone[nIdxScan] := TRUE;
				GVL_DALI.arrbBlockDTR[DALI_LINE_NUM]:= FALSE;
			ELSE
				arrInitErr[nIdxScan] := TRUE;
				GVL_DALI.arrbBlockDTR[DALI_LINE_NUM]:= FALSE;
			END_IF
		END_IF
		
	fbInitTimeOut[nIdxScan](IN:=arrInitSensor[nIdxScan] AND NOT arrInitDone[nIdxScan], PT:= T#10S); 
	
	IF fbInitTimeOut[nIdxScan].Q THEN
		arrInitErr[nIdxScan] := TRUE;
		GVL_DALI.arrbBlockDTR[DALI_LINE_NUM]:= FALSE;
	END_IF
END_FOR

stPirSensorData.bPrc:= FALSE;
FOR nPirIdxOn:= 1 TO nNumberOfSensors DO
	IF arrNiko_P46xx[nPirIdxOn].bOccupied THEN
		stPirSensorData.bPrc:= TRUE;
		EXIT;
	END_IF
END_FOR

stPirSensorData.bBrightnessRead:= arrNiko_P46xx[1].bReadingBrightness OR arrNiko_P46xx[2].bReadingBrightness OR arrNiko_P46xx[3].bReadingBrightness OR arrNiko_P46xx[4].bReadingBrightness OR arrNiko_P46xx[5].bReadingBrightness OR arrNiko_P46xx[6].bReadingBrightness;

fBrightness_1:= F_fScale(0, arrSensorScales[1].fReadMaxSensor, 0, arrSensorScales[1].fMeassureMaxSensor, 0, arrNiko_P46xx[1].nBrightnessLevel);
fBrightness_2:= F_fScale(0, arrSensorScales[2].fReadMaxSensor, 0, arrSensorScales[2].fMeassureMaxSensor, 0, arrNiko_P46xx[2].nBrightnessLevel);
fBrightness_3:= F_fScale(0, arrSensorScales[3].fReadMaxSensor, 0, arrSensorScales[3].fMeassureMaxSensor, 0, arrNiko_P46xx[3].nBrightnessLevel);
fBrightness_4:= F_fScale(0, arrSensorScales[4].fReadMaxSensor, 0, arrSensorScales[4].fMeassureMaxSensor, 0, arrNiko_P46xx[4].nBrightnessLevel);
fBrightness_5:= F_fScale(0, arrSensorScales[5].fReadMaxSensor, 0, arrSensorScales[5].fMeassureMaxSensor, 0, arrNiko_P46xx[5].nBrightnessLevel);
fBrightness_6:= F_fScale(0, arrSensorScales[6].fReadMaxSensor, 0, arrSensorScales[6].fMeassureMaxSensor, 0, arrNiko_P46xx[6].nBrightnessLevel);


IF fBrightness_1 <> 0 THEN
	stPirSensorData.fBrightness:= fBrightness_1;
END_IF
IF fBrightness_2 <> 0 THEN
	stPirSensorData.fBrightness:= MIN(fBrightness_2, stPirSensorData.fBrightness);
END_IF
IF fBrightness_3 <> 0 THEN
	stPirSensorData.fBrightness:=  MIN(fBrightness_3, stPirSensorData.fBrightness);
END_IF
IF fBrightness_4 <> 0 THEN
	stPirSensorData.fBrightness:=  MIN(fBrightness_4, stPirSensorData.fBrightness);
END_IF
IF fBrightness_5 <> 0 THEN
	stPirSensorData.fBrightness:=  MIN(fBrightness_5, stPirSensorData.fBrightness);
END_IF
IF fBrightness_6 <> 0 THEN
	stPirSensorData.fBrightness:=  MIN(fBrightness_6, stPirSensorData.fBrightness);
END_IF


IF NOT bInitialize THEN
	FOR nIdxScan := 1 TO nNumberOfSensors DO
		fbInitTimeOut[nIdxScan](IN:= FALSE);
		arrInitDone[nIdxScan] := FALSE;
		arrInitErr[nIdxScan] := FALSE;
	END_FOR
END_IF
END_ACTION

END_FUNCTION_BLOCK

// POUs/DALI/DALI_Devices/NIKO/FB_NIKO_P46xx_7Pcs
FUNCTION_BLOCK FB_NIKO_P46xx_7Pcs
VAR_INPUT
	arrShrtAdr					: ARRAY [1..7] OF BYTE;
	bInitialize					: BOOL := TRUE;
	ipCommunication				: I_DALICommunication;
	DALI_LINE_NUM				: INT := 1;	
END_VAR
VAR_OUTPUT
	arrInitErr: ARRAY [1.. nNumberOfSensors] OF BOOL;
	arrInitDone: ARRAY [1.. nNumberOfSensors] OF BOOL;
END_VAR
VAR
	arrNiko_P46xx				: ARRAY [1.. nNumberOfSensors] OF FB_DALI_Niko_P46LR(0);
	
	arrDelaySetupDALIDevice		: ARRAY [1.. nNumberOfSensors] Of TON;
	arrtDelayTime				: ARRAY [1.. nNumberOfSensors] OF TIME;
	arrInitSensor				: ARRAY [1.. nNumberOfSensors] OF BOOL;
	arrInitDone_FTrig			: ARRAY [1.. nNumberOfSensors] OF F_TRIG;
	arrInitializing				: ARRAY [1.. nNumberOfSensors] OF BOOL;
	bQueryBrightness 			: BOOL;
	bQueryOccupancy				: BOOL;
	eEventPriorityOccupancy		: E_DALIEventPriority := E_DALIEVENTPRIORITY.Middle;
	nHoldTimerOccupancy			: WORD := 5; // Value in s. 	
	nReportTimerOccupancy		: BYTE := 120; // Value in s, Preset manufacturer value
	nDeadtimeTimerOccupancy		: WORD := 100; // Value in ms, Predefined Value of DALI Standard
	bCancelHoldTimerOccupancy	: BOOL;
	nSensitivityOccupancy		: BYTE:= 3; //setting Sensivity (0..4) 0 (Off), 1 (Min), 2(Low), 3(High) and 4 (Max)

	bEnableLuxEvent				: BOOL;
	eEventPriorityBrightness	: E_DALIEventPriority := E_DALIEVENTPRIORITY.Middle;
	nDeadtimeTimerBrightness	: WORD := 1500; // Value in ms, Predefined Value of DALI Standard
	nHysteresisBrightness		: BYTE := 2; // Value in %
	nHysteresisMinBrightness	: BYTE := 10; // Absolute Value, depending on the manufacturer specific resolution
	nReportTimerBrightness		: BYTE := 120; // Value in s, Preset manufacturer value

	bAutoRead					: BOOL;
	fbAutoRequestBrightness_TON	: TOF;
	bInitTimeOut				: BOOL;
	fbInitTimeOut				: ARRAY [1.. nNumberOfSensors] OF TON;
	nIdxScan					: BYTE;
	nPirIdxOn					: BYTE;
	nBrightnessIdx				: BYTE;
	fBrightness_1				: REAL;
	fBrightness_2				: REAL;
	fBrightness_3				: REAL;
	fBrightness_4				: REAL;
	fBrightness_5				: REAL;
	fBrightness_6				: REAL;
	fBrightness_7				: REAL;
	bInitDone					: BOOL;
	bInitScalesDone				: BOOL;
	
	nCheckIdx: INT;
END_VAR
VAR_IN_OUT
	stSensorSetup 				: ST_DALI_NIKOP46SetupData ;	
	stPirSensorData				: ST_DALI_Sensor;
	arrSensorScales				: ARRAY [1.. 10] OF ST_DALI_SensorScaleMode;
END_VAR

VAR CONSTANT
	nNumberOfSensors: BYTE := 7;
END_VAR


arrNiko_P46xx[1].ipDALICommunication := ipCommunication;
arrNiko_P46xx[2].ipDALICommunication := ipCommunication;
arrNiko_P46xx[3].ipDALICommunication := ipCommunication;
arrNiko_P46xx[4].ipDALICommunication := ipCommunication;
arrNiko_P46xx[5].ipDALICommunication := ipCommunication;
arrNiko_P46xx[6].ipDALICommunication := ipCommunication;
arrNiko_P46xx[7].ipDALICommunication := ipCommunication;

IF NOT bInitScalesDone THEN
	FOR nCheckIdx:= 1 TO 10 DO
		IF arrSensorScales[nCheckIdx].fMeassureMaxSensor = 0 THEN
			arrSensorScales[nCheckIdx].fMeassureMaxSensor := 1;
		END_IF
		IF arrSensorScales[nCheckIdx].fReadMaxSensor = 0 THEN
			arrSensorScales[nCheckIdx].fReadMaxSensor := 1;
		END_IF
	END_FOR
	bInitScalesDone := TRUE;
END_IF

IF ipCommunication <> 0 THEN
	A_NIKO_P46xx();
END_IF

ACTION A_NIKO_P46xx:


FOR nIdxScan := 1 TO nNumberOfSensors DO
	//Setup parameters
		//Setup Motion part of sensor (Instance 0)
		arrNiko_P46xx[nIdxScan].eEventPriorityOccupancy:= stSensorSetup.eEventPriorityOccupancy;
		arrNiko_P46xx[nIdxScan].nHoldTimerOccupancy := stSensorSetup.nHoldTimerOccupancy ;
		arrNiko_P46xx[nIdxScan].nReportTimerOccupancy := stSensorSetup.nReportTimerOccupancy;
		arrNiko_P46xx[nIdxScan].nDeadtimeTimerOccupancy:= stSensorSetup.nDeadtimeTimerOccupancy;
		arrNiko_P46xx[nIdxScan].nSensitivityOccupancyA:= stSensorSetup.nSensitivityPIRSegmentA;
		arrNiko_P46xx[nIdxScan].nSensitivityOccupancyB:= stSensorSetup.nSensitivityPIRSegmentB;
		arrNiko_P46xx[nIdxScan].nSensitivityOccupancyC:= stSensorSetup.nSensitivityPIRSegmentC;
	
		//Setup Brightness part of sensor (Instance 1)
		arrNiko_P46xx[nIdxScan].bEnableBrightness := stSensorSetup.bEnableInstanceBrightness;
		arrNiko_P46xx[nIdxScan].eEventPriorityBrightness:= stSensorSetup.eEventPriorityBrightness;
		arrNiko_P46xx[nIdxScan].nDeadtimeTimerBrightness:= stSensorSetup.nDeadtimeTimerBrightness;
		arrNiko_P46xx[nIdxScan].nHysteresisBrightness:= stSensorSetup.nHysteresisBrightness;
		arrNiko_P46xx[nIdxScan].nHysteresisMinBrightness:= stSensorSetup.nHysteresisMinBrightness;
		arrNiko_P46xx[nIdxScan].nReportTimerBrightness:= stSensorSetup.nReportTimerBrightness;
		
	//Calculate delay time for init sensor
	arrtDelayTime[nIdxScan] := INT_TO_TIME((BYTE_TO_INT(arrShrtAdr[nIdxScan]) * 400));	
	arrDelaySetupDALIDevice[nIdxScan](IN:= bInitialize , PT:=arrtDelayTime[nIdxScan] , Q=> , ET=> );	
		
	IF arrDelaySetupDALIDevice[nIdxScan].q AND NOT GVL_DALI.arrbBlockDTR[DALI_LINE_NUM] AND NOT (arrInitDone[nIdxScan] OR arrInitErr[nIdxScan]) THEN
		arrInitSensor[nIdxScan]:= TRUE;
		GVL_DALI.arrbBlockDTR[DALI_LINE_NUM]:= TRUE;
	END_IF
	
	bQueryBrightness:= stPirSensorData.bQueryBrightness OR NOT bAutoRead;
	
	fbAutoRequestBrightness_TON(IN:= NOT fbAutoRequestBrightness_TON.Q  AND NOT stPirSensorData.bQueryBrightness , PT:= (arrtDelayTime[nIdxScan] + T#12M) , Q=>bAutoRead , ET=> );
	
	bQueryOccupancy:= NOT bAutoRead OR stPirSensorData.bQueryBrightness;
	
	arrNiko_P46xx[nIdxScan](
		bError=> , 
		ipResultMessage=> , 
		bInitialize:=  arrInitSensor[nIdxScan], 
		nShortAddress:= arrShrtAdr[nIdxScan], 
		nOptions:= , 
		bQueryOccupancy:= bQueryOccupancy, 
		bQueryBrightness:= bQueryBrightness, 
		bCancelHoldTimerOccupancy:= bCancelHoldTimerOccupancy, 
		bInitializing=> arrInitializing[nIdxScan] , 
		bReadingOccupancy=> , 
		bReadingBrightness=> , 
		bOccupied=> , 
		nBrightnessLevel=> );
	
	IF arrNiko_P46xx[nIdxScan].bError THEN
		GVL_DALI_LatestError.arrLineShrtAddr[DALI_LINE_NUM] := arrShrtAdr[nIdxScan];
	END_IF
	
	arrInitDone_FTrig[nIdxScan](CLK:=arrInitializing[nIdxScan] );	
		IF arrInitDone_FTrig[nIdxScan].Q THEN
			IF NOT bInitTimeOut THEN
				arrInitDone[nIdxScan] := TRUE;
				GVL_DALI.arrbBlockDTR[DALI_LINE_NUM]:= FALSE;
			ELSE
				arrInitErr[nIdxScan] := TRUE;
				GVL_DALI.arrbBlockDTR[DALI_LINE_NUM]:= FALSE;
			END_IF
		END_IF
		
	fbInitTimeOut[nIdxScan](IN:=arrInitSensor[nIdxScan] AND NOT arrInitDone[nIdxScan], PT:= T#10S); 
	
	IF fbInitTimeOut[nIdxScan].Q THEN
		arrInitErr[nIdxScan] := TRUE;
		GVL_DALI.arrbBlockDTR[DALI_LINE_NUM]:= FALSE;
	END_IF
END_FOR

stPirSensorData.bPrc:= FALSE;
FOR nPirIdxOn:= 1 TO nNumberOfSensors DO
	IF arrNiko_P46xx[nPirIdxOn].bOccupied THEN
		stPirSensorData.bPrc:= TRUE;
		EXIT;
	END_IF
END_FOR

stPirSensorData.bBrightnessRead:= arrNiko_P46xx[1].bReadingBrightness OR arrNiko_P46xx[2].bReadingBrightness OR arrNiko_P46xx[3].bReadingBrightness OR arrNiko_P46xx[4].bReadingBrightness OR arrNiko_P46xx[5].bReadingBrightness OR arrNiko_P46xx[6].bReadingBrightness OR arrNiko_P46xx[7].bReadingBrightness;

fBrightness_1:= F_fScale(0, arrSensorScales[1].fReadMaxSensor, 0, arrSensorScales[1].fMeassureMaxSensor, 0, arrNiko_P46xx[1].nBrightnessLevel);
fBrightness_2:= F_fScale(0, arrSensorScales[2].fReadMaxSensor, 0, arrSensorScales[2].fMeassureMaxSensor, 0, arrNiko_P46xx[2].nBrightnessLevel);
fBrightness_3:= F_fScale(0, arrSensorScales[3].fReadMaxSensor, 0, arrSensorScales[3].fMeassureMaxSensor, 0, arrNiko_P46xx[3].nBrightnessLevel);
fBrightness_4:= F_fScale(0, arrSensorScales[4].fReadMaxSensor, 0, arrSensorScales[4].fMeassureMaxSensor, 0, arrNiko_P46xx[4].nBrightnessLevel);
fBrightness_5:= F_fScale(0, arrSensorScales[5].fReadMaxSensor, 0, arrSensorScales[5].fMeassureMaxSensor, 0, arrNiko_P46xx[5].nBrightnessLevel);
fBrightness_6:= F_fScale(0, arrSensorScales[6].fReadMaxSensor, 0, arrSensorScales[6].fMeassureMaxSensor, 0, arrNiko_P46xx[6].nBrightnessLevel);
fBrightness_7:= F_fScale(0, arrSensorScales[7].fReadMaxSensor, 0, arrSensorScales[7].fMeassureMaxSensor, 0, arrNiko_P46xx[7].nBrightnessLevel);

IF fBrightness_1 <> 0 THEN
	stPirSensorData.fBrightness:= fBrightness_1;
END_IF
IF fBrightness_2 <> 0 THEN
	stPirSensorData.fBrightness:= MIN(fBrightness_2, stPirSensorData.fBrightness);
END_IF
IF fBrightness_3 <> 0 THEN
	stPirSensorData.fBrightness:=  MIN(fBrightness_3, stPirSensorData.fBrightness);
END_IF
IF fBrightness_4 <> 0 THEN
	stPirSensorData.fBrightness:=  MIN(fBrightness_4, stPirSensorData.fBrightness);
END_IF
IF fBrightness_5 <> 0 THEN
	stPirSensorData.fBrightness:=  MIN(fBrightness_5, stPirSensorData.fBrightness);
END_IF
IF fBrightness_6 <> 0 THEN
	stPirSensorData.fBrightness:=  MIN(fBrightness_6, stPirSensorData.fBrightness);
END_IF
IF fBrightness_7 <> 0 THEN
	stPirSensorData.fBrightness:=  MIN(fBrightness_7, stPirSensorData.fBrightness);
END_IF


IF NOT bInitialize THEN
	FOR nIdxScan := 1 TO nNumberOfSensors DO
		fbInitTimeOut[nIdxScan](IN:= FALSE);
		arrInitDone[nIdxScan] := FALSE;
		arrInitErr[nIdxScan] := FALSE;
	END_FOR
END_IF
END_ACTION

END_FUNCTION_BLOCK

// POUs/DALI/DALI_Devices/NIKO/FB_NIKO_P46xx_8Pcs
FUNCTION_BLOCK FB_NIKO_P46xx_8Pcs
VAR_INPUT
	arrShrtAdr					: ARRAY [1..8] OF BYTE;
	bInitialize					: BOOL := TRUE;
	ipCommunication				: I_DALICommunication;
	DALI_LINE_NUM				: INT := 1;	
END_VAR
VAR_OUTPUT
	arrInitErr: ARRAY [1.. nNumberOfSensors] OF BOOL;
	arrInitDone: ARRAY [1.. nNumberOfSensors] OF BOOL;
END_VAR
VAR
	arrNiko_P46xx				: ARRAY [1.. nNumberOfSensors] OF FB_DALI_Niko_P46LR(0);
	
	arrDelaySetupDALIDevice		: ARRAY [1.. nNumberOfSensors] Of TON;
	arrtDelayTime				: ARRAY [1.. nNumberOfSensors] OF TIME;
	arrInitSensor				: ARRAY [1.. nNumberOfSensors] OF BOOL;
	arrInitDone_FTrig			: ARRAY [1.. nNumberOfSensors] OF F_TRIG;
	arrInitializing				: ARRAY [1.. nNumberOfSensors] OF BOOL;
	bQueryBrightness 			: BOOL;
	bQueryOccupancy				: BOOL;
	eEventPriorityOccupancy		: E_DALIEventPriority := E_DALIEVENTPRIORITY.Middle;
	nHoldTimerOccupancy			: WORD := 5; // Value in s. 	
	nReportTimerOccupancy		: BYTE := 120; // Value in s, Preset manufacturer value
	nDeadtimeTimerOccupancy		: WORD := 100; // Value in ms, Predefined Value of DALI Standard
	bCancelHoldTimerOccupancy	: BOOL;
	nSensitivityOccupancy		: BYTE:= 3; //setting Sensivity (0..4) 0 (Off), 1 (Min), 2(Low), 3(High) and 4 (Max)

	bEnableLuxEvent				: BOOL;
	eEventPriorityBrightness	: E_DALIEventPriority := E_DALIEVENTPRIORITY.Middle;
	nDeadtimeTimerBrightness	: WORD := 1500; // Value in ms, Predefined Value of DALI Standard
	nHysteresisBrightness		: BYTE := 2; // Value in %
	nHysteresisMinBrightness	: BYTE := 10; // Absolute Value, depending on the manufacturer specific resolution
	nReportTimerBrightness		: BYTE := 120; // Value in s, Preset manufacturer value

	bAutoRead					: BOOL;
	fbAutoRequestBrightness_TON	: TOF;
	bInitTimeOut				: BOOL;
	fbInitTimeOut				: ARRAY [1.. nNumberOfSensors] OF TON;
	nIdxScan					: BYTE;
	nPirIdxOn					: BYTE;
	nBrightnessIdx				: BYTE;
	fBrightness_1				: REAL;
	fBrightness_2				: REAL;
	fBrightness_3				: REAL;
	fBrightness_4				: REAL;
	fBrightness_5				: REAL;
	fBrightness_6				: REAL;
	fBrightness_7				: REAL;
	fBrightness_8				: REAL;
	bInitDone					: BOOL;
	bInitScalesDone				: BOOL;
	
	nCheckIdx: INT;
END_VAR
VAR_IN_OUT
	stSensorSetup 				: ST_DALI_NIKOP46SetupData ;	
	stPirSensorData				: ST_DALI_Sensor;
	arrSensorScales				: ARRAY [1..10] OF ST_DALI_SensorScaleMode;
END_VAR

VAR CONSTANT
	nNumberOfSensors: BYTE := 8;
END_VAR


arrNiko_P46xx[1].ipDALICommunication := ipCommunication;
arrNiko_P46xx[2].ipDALICommunication := ipCommunication;
arrNiko_P46xx[3].ipDALICommunication := ipCommunication;
arrNiko_P46xx[4].ipDALICommunication := ipCommunication;
arrNiko_P46xx[5].ipDALICommunication := ipCommunication;
arrNiko_P46xx[6].ipDALICommunication := ipCommunication;
arrNiko_P46xx[7].ipDALICommunication := ipCommunication;
arrNiko_P46xx[8].ipDALICommunication := ipCommunication;

IF NOT bInitScalesDone THEN
	FOR nCheckIdx:= 1 TO 8 DO
		IF arrSensorScales[nCheckIdx].fMeassureMaxSensor = 0 THEN
			arrSensorScales[nCheckIdx].fMeassureMaxSensor := 1;
		END_IF
		IF arrSensorScales[nCheckIdx].fReadMaxSensor = 0 THEN
			arrSensorScales[nCheckIdx].fReadMaxSensor := 1;
		END_IF
	END_FOR
	bInitScalesDone := TRUE;
END_IF

IF ipCommunication <> 0 THEN
	A_NIKO_P46xx();
END_IF

ACTION A_NIKO_P46xx:


FOR nIdxScan := 1 TO nNumberOfSensors DO
	//Setup parameters
		//Setup Motion part of sensor (Instance 0)
		arrNiko_P46xx[nIdxScan].eEventPriorityOccupancy:= stSensorSetup.eEventPriorityOccupancy;
		arrNiko_P46xx[nIdxScan].nHoldTimerOccupancy := stSensorSetup.nHoldTimerOccupancy ;
		arrNiko_P46xx[nIdxScan].nReportTimerOccupancy := stSensorSetup.nReportTimerOccupancy;
		arrNiko_P46xx[nIdxScan].nDeadtimeTimerOccupancy:= stSensorSetup.nDeadtimeTimerOccupancy;
		arrNiko_P46xx[nIdxScan].nSensitivityOccupancyA:= stSensorSetup.nSensitivityPIRSegmentA;
		arrNiko_P46xx[nIdxScan].nSensitivityOccupancyB:= stSensorSetup.nSensitivityPIRSegmentB;
		arrNiko_P46xx[nIdxScan].nSensitivityOccupancyC:= stSensorSetup.nSensitivityPIRSegmentC;
	
		//Setup Brightness part of sensor (Instance 1)
		arrNiko_P46xx[nIdxScan].bEnableBrightness := stSensorSetup.bEnableInstanceBrightness;
		arrNiko_P46xx[nIdxScan].eEventPriorityBrightness:= stSensorSetup.eEventPriorityBrightness;
		arrNiko_P46xx[nIdxScan].nDeadtimeTimerBrightness:= stSensorSetup.nDeadtimeTimerBrightness;
		arrNiko_P46xx[nIdxScan].nHysteresisBrightness:= stSensorSetup.nHysteresisBrightness;
		arrNiko_P46xx[nIdxScan].nHysteresisMinBrightness:= stSensorSetup.nHysteresisMinBrightness;
		arrNiko_P46xx[nIdxScan].nReportTimerBrightness:= stSensorSetup.nReportTimerBrightness;
		
	//Calculate delay time for init sensor
	arrtDelayTime[nIdxScan] := INT_TO_TIME((BYTE_TO_INT(arrShrtAdr[nIdxScan]) * 400));	
	arrDelaySetupDALIDevice[nIdxScan](IN:= bInitialize , PT:=arrtDelayTime[nIdxScan] , Q=> , ET=> );	
		
	IF arrDelaySetupDALIDevice[nIdxScan].q AND NOT GVL_DALI.arrbBlockDTR[DALI_LINE_NUM] AND NOT (arrInitDone[nIdxScan] OR arrInitErr[nIdxScan]) THEN
		arrInitSensor[nIdxScan]:= TRUE;
		GVL_DALI.arrbBlockDTR[DALI_LINE_NUM]:= TRUE;
	END_IF
	
	bQueryBrightness:= stPirSensorData.bQueryBrightness OR NOT bAutoRead;
	
	fbAutoRequestBrightness_TON(IN:= NOT fbAutoRequestBrightness_TON.Q  AND NOT stPirSensorData.bQueryBrightness , PT:= (arrtDelayTime[nIdxScan] + T#12M) , Q=>bAutoRead , ET=> );
	
	bQueryOccupancy:= NOT bAutoRead OR stPirSensorData.bQueryBrightness;
	
	arrNiko_P46xx[nIdxScan](
		bError=> , 
		ipResultMessage=> , 
		bInitialize:=  arrInitSensor[nIdxScan], 
		nShortAddress:= arrShrtAdr[nIdxScan], 
		nOptions:= , 
		bQueryOccupancy:= bQueryOccupancy, 
		bQueryBrightness:= bQueryBrightness, 
		bCancelHoldTimerOccupancy:= bCancelHoldTimerOccupancy, 
		bInitializing=> arrInitializing[nIdxScan] , 
		bReadingOccupancy=> , 
		bReadingBrightness=> , 
		bOccupied=> , 
		nBrightnessLevel=> );
	
	IF arrNiko_P46xx[nIdxScan].bError THEN
		GVL_DALI_LatestError.arrLineShrtAddr[DALI_LINE_NUM] :=arrShrtAdr[nIdxScan];
	END_IF
	
	arrInitDone_FTrig[nIdxScan](CLK:=arrInitializing[nIdxScan] );	
		IF arrInitDone_FTrig[nIdxScan].Q THEN
			IF NOT bInitTimeOut THEN
				arrInitDone[nIdxScan] := TRUE;
				GVL_DALI.arrbBlockDTR[DALI_LINE_NUM]:= FALSE;
			ELSE
				arrInitErr[nIdxScan] := TRUE;
				GVL_DALI.arrbBlockDTR[DALI_LINE_NUM]:= FALSE;
			END_IF
		END_IF
		
	fbInitTimeOut[nIdxScan](IN:=arrInitSensor[nIdxScan] AND NOT arrInitDone[nIdxScan], PT:= T#10S); 
	
	IF fbInitTimeOut[nIdxScan].Q THEN
		arrInitErr[nIdxScan] := TRUE;
		GVL_DALI.arrbBlockDTR[DALI_LINE_NUM]:= FALSE;
	END_IF
END_FOR

stPirSensorData.bPrc:= FALSE;
FOR nPirIdxOn:= 1 TO nNumberOfSensors DO
	IF arrNiko_P46xx[nPirIdxOn].bOccupied THEN
		stPirSensorData.bPrc:= TRUE;
		EXIT;
	END_IF
END_FOR

stPirSensorData.bBrightnessRead:=	arrNiko_P46xx[1].bReadingBrightness OR arrNiko_P46xx[2].bReadingBrightness OR arrNiko_P46xx[3].bReadingBrightness OR arrNiko_P46xx[4].bReadingBrightness OR arrNiko_P46xx[5].bReadingBrightness OR
														arrNiko_P46xx[6].bReadingBrightness OR arrNiko_P46xx[7].bReadingBrightness OR arrNiko_P46xx[8].bReadingBrightness;

fBrightness_1:= F_fScale(0, arrSensorScales[1].fReadMaxSensor, 0, arrSensorScales[1].fMeassureMaxSensor, 0, arrNiko_P46xx[1].nBrightnessLevel);
fBrightness_2:= F_fScale(0, arrSensorScales[2].fReadMaxSensor, 0, arrSensorScales[2].fMeassureMaxSensor, 0, arrNiko_P46xx[2].nBrightnessLevel);
fBrightness_3:= F_fScale(0, arrSensorScales[3].fReadMaxSensor, 0, arrSensorScales[3].fMeassureMaxSensor, 0, arrNiko_P46xx[3].nBrightnessLevel);
fBrightness_4:= F_fScale(0, arrSensorScales[4].fReadMaxSensor, 0, arrSensorScales[4].fMeassureMaxSensor, 0, arrNiko_P46xx[4].nBrightnessLevel);
fBrightness_5:= F_fScale(0, arrSensorScales[5].fReadMaxSensor, 0, arrSensorScales[5].fMeassureMaxSensor, 0, arrNiko_P46xx[5].nBrightnessLevel);
fBrightness_6:= F_fScale(0, arrSensorScales[6].fReadMaxSensor, 0, arrSensorScales[6].fMeassureMaxSensor, 0, arrNiko_P46xx[6].nBrightnessLevel);
fBrightness_7:= F_fScale(0, arrSensorScales[7].fReadMaxSensor, 0, arrSensorScales[7].fMeassureMaxSensor, 0, arrNiko_P46xx[7].nBrightnessLevel);
fBrightness_8:= F_fScale(0, arrSensorScales[8].fReadMaxSensor, 0, arrSensorScales[8].fMeassureMaxSensor, 0, arrNiko_P46xx[8].nBrightnessLevel);


IF fBrightness_1 <> 0 THEN
	stPirSensorData.fBrightness:= fBrightness_1;
END_IF
IF fBrightness_2 <> 0 THEN
	stPirSensorData.fBrightness:= MIN(fBrightness_2, stPirSensorData.fBrightness);
END_IF
IF fBrightness_3 <> 0 THEN
	stPirSensorData.fBrightness:=  MIN(fBrightness_3, stPirSensorData.fBrightness);
END_IF
IF fBrightness_4 <> 0 THEN
	stPirSensorData.fBrightness:=  MIN(fBrightness_4, stPirSensorData.fBrightness);
END_IF
IF fBrightness_5 <> 0 THEN
	stPirSensorData.fBrightness:=  MIN(fBrightness_5, stPirSensorData.fBrightness);
END_IF
IF fBrightness_6 <> 0 THEN
	stPirSensorData.fBrightness:= MIN(fBrightness_6, stPirSensorData.fBrightness);
END_IF
IF fBrightness_7 <> 0 THEN
	stPirSensorData.fBrightness:=  MIN(fBrightness_7, stPirSensorData.fBrightness);
END_IF
IF fBrightness_8 <> 0 THEN
	stPirSensorData.fBrightness:=  MIN(fBrightness_8, stPirSensorData.fBrightness);
END_IF


IF NOT bInitialize THEN
	FOR nIdxScan := 1 TO nNumberOfSensors DO
		fbInitTimeOut[nIdxScan](IN:= FALSE);
		arrInitDone[nIdxScan] := FALSE;
		arrInitErr[nIdxScan] := FALSE;
	END_FOR
END_IF
END_ACTION

END_FUNCTION_BLOCK

// POUs/DALI/DALI_Devices/NIKO/FB_NIKO_P46xx_9Pcs
FUNCTION_BLOCK FB_NIKO_P46xx_9Pcs
VAR_INPUT
	arrShrtAdr					: ARRAY [1..9] OF BYTE;
	bInitialize					: BOOL := TRUE;
	ipCommunication				: I_DALICommunication;
	DALI_LINE_NUM				: INT := 1;	
END_VAR
VAR_OUTPUT
	arrInitErr: ARRAY [1.. nNumberOfSensors] OF BOOL;
	arrInitDone: ARRAY [1.. nNumberOfSensors] OF BOOL;
END_VAR
VAR
	arrNiko_P46xx				: ARRAY [1.. nNumberOfSensors] OF FB_DALI_Niko_P46LR(0);
	
	arrDelaySetupDALIDevice		: ARRAY [1.. nNumberOfSensors] Of TON;
	arrtDelayTime				: ARRAY [1.. nNumberOfSensors] OF TIME;
	arrInitSensor				: ARRAY [1.. nNumberOfSensors] OF BOOL;
	arrInitDone_FTrig			: ARRAY [1.. nNumberOfSensors] OF F_TRIG;
	arrInitializing				: ARRAY [1.. nNumberOfSensors] OF BOOL;
	bQueryBrightness 			: BOOL;
	bQueryOccupancy				: BOOL;
	eEventPriorityOccupancy		: E_DALIEventPriority := E_DALIEVENTPRIORITY.Middle;
	nHoldTimerOccupancy			: WORD := 5; // Value in s. 	
	nReportTimerOccupancy		: BYTE := 120; // Value in s, Preset manufacturer value
	nDeadtimeTimerOccupancy		: WORD := 100; // Value in ms, Predefined Value of DALI Standard
	bCancelHoldTimerOccupancy	: BOOL;
	nSensitivityOccupancy		: BYTE:= 3; //setting Sensivity (0..4) 0 (Off), 1 (Min), 2(Low), 3(High) and 4 (Max)

	bEnableLuxEvent				: BOOL;
	eEventPriorityBrightness	: E_DALIEventPriority := E_DALIEVENTPRIORITY.Middle;
	nDeadtimeTimerBrightness	: WORD := 1500; // Value in ms, Predefined Value of DALI Standard
	nHysteresisBrightness		: BYTE := 2; // Value in %
	nHysteresisMinBrightness	: BYTE := 10; // Absolute Value, depending on the manufacturer specific resolution
	nReportTimerBrightness		: BYTE := 120; // Value in s, Preset manufacturer value

	bAutoRead					: BOOL;
	fbAutoRequestBrightness_TON	: TOF;
	bInitTimeOut				: BOOL;
	fbInitTimeOut				: ARRAY [1.. nNumberOfSensors] OF TON;
	nIdxScan					: BYTE;
	nPirIdxOn					: BYTE;
	nBrightnessIdx				: BYTE;
	fBrightness_1				: REAL;
	fBrightness_2				: REAL;
	fBrightness_3				: REAL;
	fBrightness_4				: REAL;
	fBrightness_5				: REAL;
	fBrightness_6				: REAL;
	fBrightness_7				: REAL;
	fBrightness_8				: REAL;
	fBrightness_9				: REAL;
	bInitDone					: BOOL;
	bInitScalesDone				: BOOL;
	
	nCheckIdx: INT;
END_VAR
VAR_IN_OUT
	stSensorSetup 				: ST_DALI_NIKOP46SetupData ;	
	stPirSensorData				: ST_DALI_Sensor;
	arrSensorScales				: ARRAY [1..10] OF ST_DALI_SensorScaleMode;
END_VAR

VAR CONSTANT
	nNumberOfSensors: BYTE := 9;
END_VAR


arrNiko_P46xx[1].ipDALICommunication := ipCommunication;
arrNiko_P46xx[2].ipDALICommunication := ipCommunication;
arrNiko_P46xx[3].ipDALICommunication := ipCommunication;
arrNiko_P46xx[4].ipDALICommunication := ipCommunication;
arrNiko_P46xx[5].ipDALICommunication := ipCommunication;
arrNiko_P46xx[6].ipDALICommunication := ipCommunication;
arrNiko_P46xx[7].ipDALICommunication := ipCommunication;
arrNiko_P46xx[8].ipDALICommunication := ipCommunication;
arrNiko_P46xx[9].ipDALICommunication := ipCommunication;

IF NOT bInitScalesDone THEN
	FOR nCheckIdx:= 1 TO 9 DO
		IF arrSensorScales[nCheckIdx].fMeassureMaxSensor = 0 THEN
			arrSensorScales[nCheckIdx].fMeassureMaxSensor := 1;
		END_IF
		IF arrSensorScales[nCheckIdx].fReadMaxSensor = 0 THEN
			arrSensorScales[nCheckIdx].fReadMaxSensor := 1;
		END_IF
	END_FOR
	bInitScalesDone := TRUE;
END_IF

IF ipCommunication <> 0 THEN
	A_NIKO_P46xx();
END_IF

ACTION A_NIKO_P46xx:


